# B&R Automation Studio project ABC_Pltzr
Automation Studio 

## Configuration PPC70_JOB24025

### Config.mpfilemanagerui - 4PPC70_101G_20F005/mapp/Config.mpfilemanagerui
```
Element gMpLinkMpFileManagerUI (Type=mpfilemanagerui)
```

## Logical view

Binary libraries used (declarations not repeated): AsBrStr, AsTCP, FileIO

### 1stReadme-ConfigAndRecipes.txt
```
Package name:
=============
appConfigAndRecipes

Desription:
===========
Package contains support for application wide Configuration and Recipe handling.

About:
======

Dependencies:
=============
- B&R Libraries: FileIO
- Other: bglib C utilities

Usage:
======
IMPORTANT: Make sure that the package is always located as a LAST item in the logical view!!!
This limitation is due to the compilatoin dependency and references to user defined structures defined
elsewhere and utilized here.

Examples:
=============
TODO
```

### MachineIO.typ
```iecst
(********************************************************************

 * COPYRIGHT -- Piedmont Automation Inc.

 ********************************************************************

 * File: MachineIO.typ

 * Author: goran

 * Created: Jun 1, 2015

 ********************************************************************

 *)
(*********************************************************************************

Machine IO Structure

*********************************************************************************)

TYPE
	machineIO_typ : 	STRUCT
		din : machineDI_typ;
		dout : machineDO_typ;
	END_STRUCT;
END_TYPE

(*********************************************************************************

	Machine Digital Inputs

*********************************************************************************)

TYPE
	machineDI_typ : 	STRUCT
		MCR : BOOL; (*Master Control Relay Energized*)
		Guard_DS1 : BOOL; (*Guard 1 Open DS1 # GUARD DOOR INSERTER*)
		Guard_DS2 : BOOL; (*Guard 2 Open DS2 # GUARD DOOR GROUPING RIGHT*)
		Guard_DS3 : BOOL; (*Guard 3 Open DS3 # GUARD DOOR DISPENSER*)
		Guard_DS4 : BOOL; (*Guard 4 Open DS4 # GUARD DOOR GROUPING LEFT*)
		Guard_DS5 : BOOL; (*Guard 5 Open DS5 # TBD*)
		Guard_DS6 : BOOL; (*Guard 6 Open DS6 # TBD*)
		EStop_PB1 : BOOL; (*EStop status 1 - PB1 - Enclosure*)
		EStop_PB2 : BOOL; (*EStop status 2 - PB2 - Infeed*)
		EStop_PB3 : BOOL; (*EStop status 3 - PB3 - Dispenser*)
		EStop_PB4 : BOOL; (*EStop status 4 - PB 4 - HMI*)
		EStop_PB5 : BOOL; (*EStop status 5 - PB5 - TBD*)
		EStop_PB6 : BOOL; (*EStop status 6 - PB6 - TBD*)
		MotorOverloads_OL : BOOL; (*MotorOverloads*)
		CustomerDischargeEnable_CR6 : BOOL; (*Customer Discharge Enable*)
		AirPressureSwitch_APS : BOOL; (*Air Pressure Switch APS*)
		PalletMagazineControl_SS2 : BOOL; (*Pallet Dispenser in Run Mode SS2*)
		PalleteDischLightCurtain_OSSD1 : BOOL; (*Pallete Dispenser Light Curtain CH A*)
		PalleteDischLightCurtain_OSSD2 : BOOL; (*Pallete Dispenser Light Curtain CH B*)
		ElevatorDetectPalletLayerLF_EE1 : BOOL; (*Detect Layer On Pallet EE1*)
		ProductAtStage_EE4Phy : BOOL;
		ProductAtStage_EE4TmrOn : TON;
		ProductAtStage_EE4TmrOf : TOF;
		ProductAtStage_EE4 : BOOL; (*Product/Case at Stage Position*)
		ElevatorDetectPalletLayerRT_EE3 : BOOL; (*Detect Layer On Pallet 2nd Eye EE3*)
		ZZZZZZZZZZZZZZZZZZZZZZZZZZZ : USINT;
		ElevatorFullUp_PR1 : BOOL; (*Elevator Full Up PR1*)
		ElevatorFullDown_PR2 : BOOL; (*Elevator Full Down PR2*)
		ElevatorAtGroupingRaise_PR4 : BOOL; (*Elevator @ Level for Raise PR4*)
		ElevatorAtGroupingLower_PR3 : BOOL; (*Elevator @ Level for Lower PR3*)
		ElevatorStopBlockRT_PR34 : BOOL; (*Elevator Stop Block Right Is Clear PR34*)
		ElevatorStopBlockLF_PR33 : BOOL; (*Elevator Stop Block Left Is Clear PR33*)
		ElevatorChainSlackRT_LS8 : BOOL; (*Elevator Chain Slack Right LS8*)
		ElevatorChainSlackLF_LS7 : BOOL; (*Elevator Chain Slack Left LS7*)
		TransferTableAtGrouping_PR6 : BOOL; (*Transfer Table At Grouping Side PR6*)
		TransferTableAtPallete_PR5 : BOOL; (*Table at Pallet Side PR5*)
		LayerStopBarDown_PR8 : BOOL; (*Layer Stop Bar/Stripper Bar is Down PR8*)
		LayerStopBarUp_PR7 : BOOL; (*Layer Stop Bar/Stripper Bar is Up PR7*)
		ProductAtInfeed_EE2Phy : BOOL; (*Product At Infeed Case / Counter EE2*)
		ProductAtInfeed_EE2TmrOn : TON; (*Product At Infeed Case / Counter EE2*)
		ProductAtInfeed_EE2TmrOf : TOF; (*Product At Infeed Case / Counter EE2*)
		ProductAtInfeed_EE2 : BOOL; (*Product At Infeed Case / Counter EE2*)
		RowTooLong_EE8Phy : BOOL;
		RowTooLong_EE8TmrOn : TON;
		RowTooLong_EE8TmrOf : TOF;
		RowTooLong_EE8 : BOOL; (*Comparison Count Row Too Long EE8*)
		RowPusherAtElevator_PR13 : BOOL; (*Row Pusher At Elevator PR13*)
		RowPusherReturned_PR11 : BOOL; (*Row Pusher Returned PR11*)
		PalletClawsAtTop_PR14 : BOOL; (*Pallet Dispenser at Top Position PR14*)
		PalletClawsAtMiddleLow_PR15 : BOOL; (*Pallet Dispenser Claws at Middle Position PR15*)
		PalletClawsAtMiddleHi_PR15A : BOOL; (*Pallet Claws at upper Middle*)
		PalletClawsAtBottom_PR16 : BOOL; (*Pallet Dispenser Claws at Bottom Position PR16*)
		PalletClawsClosedRT_PR18 : BOOL; (*Pallet Dispenser Right Claw Closed PR18*)
		PalletClawsClosedLF_PR20 : BOOL; (*Pallet Dispenser Left Claw Closed PR20*)
		PalletDispenserLowSupply_EE7 : BOOL; (*Pallet Dispenser Low Pallet Supply EE7*)
		PalletDispenserChainSlack_PR21 : BOOL; (*Pallet Dispenser Chain Slack PR21*)
		PalletDownOnDispenserCV_EE9 : BOOL; (*Pallet Dispenser Down on Dispenser Conveyor EE9*)
		ZZZZZZZZZZZZZZZZZZZZZZZZZZZ1 : USINT;
		Reset_PB : BOOL; (*Reset PushButton PB6*)
		PalletAtMachine_EE12 : BOOL; (*PalletAtMachine*)
		PalletAtDischarge_EE16 : BOOL; (*PalletAtDischarge*)
		Inserter_Control_In_Run_Mode : BOOL; (*Inserter Control in Run Mode SS3*)
		Inserter_Guard_Eye : BOOL; (*Inserter Guard Eye EE30*)
		Discharge_Guard_Eye : BOOL; (*Discharge Guard Eye EE5*)
		Pallet_On_Conveyor_2_After : BOOL; (*Pallet On Conveyor 2 After EE17*)
		Pallet_On_Conveyor_1_After : BOOL; (*Pallet On Conveyor 1 After EE16*)
		Drive1_Running : BOOL; (*Drive 1 Running VFD1*)
		Drive4_OverCurrent : BOOL; (*Drive 4 OverCurrent VFD4*)
		Motor_Protectors : BOOL; (*Motor Protectors OL*)
		Row_Pusher_At_PreGrouping : BOOL; (*Row Pusher At PreGrouping PR12*)
		Row_Pusher_Is_Down : BOOL; (*Row Pusher Is Down PR10*)
		Row_Pusher_Is_Up : BOOL; (*Row Pusher Is Up PR9*)
		MACHINE_ESTOPS_OK : BOOL; (*Machine ESTOPS*)
		ESTOPS_OK : BOOL; (*E-STOPS OKAY PB1*)
		Pallet_Chains_Are_Up : BOOL; (*Pallet Chains Are Up PR35*)
		Turn_Table_Is_Up_NOP : BOOL; (* TurnTable is Up-NOP PR23*)
		Turn_Table_Is_Down : BOOL; (* TurnTable is Down PR22*)
		Screen_Access : BOOL; (*Screen Access SS1*)
		AuxVFDsOk : BOOL; (*Auxiliar VFD's OK*)
		InserterAtMagazine : BOOL; (*Inserter At Magazine PR28*)
		InserterVacuumCupsIsDown : BOOL; (*Inserter Vacuum Cups Is Down PR27*)
		InserterIsDown : BOOL; (*Inserter is Down PR29*)
		InserterTierSheetBeltSlack : BOOL; (*Inserter Tier Sheet Belt Slack *)
		InserterLowTierSheetLevel : BOOL; (*Low Tier Sheet Level EE10*)
		InserterIsUp : BOOL; (*Inserter is Up PR26*)
		InserterSheetHeld : BOOL; (*Inserter Tier Sheet Held EE15*)
		Turn_Table_CW_Stop_Position : BOOL; (*Turn Table CW Stop Position PR24*)
	END_STRUCT;
END_TYPE

(*********************************************************************************

	Machine Digital Outputs

*********************************************************************************)

TYPE
	machineDO_typ : 	STRUCT
		MachineFaultBeacon_LT1 : BOOL; (*Machine Fault Beacon LT1*)
		MachineOkBeacon_LT2 : BOOL; (*Machine OK Beacon LT2*)
		PalletLowSupplyBeacon_LT3 : BOOL; (*Pallet Low Supply Beacon Light LT3*)
		LayerStopBarRaise_M3F : BOOL; (*Layer Bar Raise M3F*)
		LayerStopBarLower_M3R : BOOL; (*Layer Bar Lower M3R*)
		RowFormingRollers_M5 : BOOL; (*Grouping Rollers M5*)
		ProductInfeedCV_M6 : BOOL; (*Product Infeed Belt M6*)
		PalletDispenserCV_M7 : BOOL; (*Pallet Dispenser Conveyor M7*)
		PalletDispenserRaise_M8F : BOOL; (*Pallet Dispenser Raise M8F*)
		PalletDispenserLower_M8R : BOOL; (*Pallet Dispenser Lower M8R*)
		CustomerMachineRunning_CR4 : BOOL; (*Customer Facing Machine Running CR4*)
		CustomerMachineRunning_CR5 : BOOL; (*Customer Facing Machine Running CR5*)
		AirDump_SOL0 : BOOL; (*Air Dump SOL0*)
		TransferTableToGrouping_M2R : BOOL; (*Transfer Table To Grouping M2R*)
		TransferTableToPallet_M2F : BOOL; (*Transfer Table To Pallet M2F*)
		RowPusherReturn_M4R : BOOL; (*VFD4 REV*)
		RowPusherForward_M4F : BOOL; (*VFD4 FWD*)
		PalletClawsOpen_SOL7B : BOOL; (*Open Pallet Dispenser Claws SOL7B*)
		PalletClawsClose_SOL7A : BOOL; (*Close Pallet Dispenser Claws SOL7A*)
		FrontSquaringRetract_SOL11B : BOOL; (*End/Front Squaring Retract SOL11B*)
		FrontSquaringExtend_SOL11A : BOOL; (*End/Front Squaring Extend SOL11A*)
		SideSquaringRetract_SOL8B : BOOL; (*Side Squaring Retract SOL8B*)
		SideSquaringExtend_SOL8A : BOOL; (*Side Squaring Extend SOL8A*)
		BladeStop1Up_SOL3A : BOOL; (*Blade Stop 1 Lower SOL3B*)
		BladeStop1Dw_SOL3B : BOOL; (*Blade Stop 1 Raise SOL3A*)
		BladeStop2Up_SOL4A : BOOL; (*Blade Stop 1 Lower SOL3B*)
		BladeStop2Dw_SOL4B : BOOL; (*Blade Stop 1 Raise SOL3A*)
		BladeStop3Up_SOL5A : BOOL; (*Blade Stop 1 Lower SOL3B*)
		BladeStop3Dw_SOL5B : BOOL; (*Blade Stop 1 Raise SOL3A*)
		BladeStop4Up_SOL6A : BOOL; (*Blade Stop 1 Lower SOL3B*)
		BladeStop4Dw_SOL6B : BOOL; (*Blade Stop 1 Raise SOL3A*)
		BladeStop5Up_SOL13A : BOOL; (*Blade Stop 1 Lower SOL3B*)
		BladeStop5Dw_SOL13B : BOOL; (*Blade Stop 1 Raise SOL3A*)
		BladeStop6Up_SOL14A : BOOL; (*Blade Stop 1 Lower SOL3B*)
		BladeStop6Dw_SOL14B : BOOL; (*Blade Stop 1 Raise SOL3A*)
		CaseTurnerLower_SOL2B : BOOL; (*Case Turner Lower SOL2B*)
		CaseTurnerRaise_SOL2A : BOOL; (*Case Turner Raise SOL2A*)
		ZZZZZZZZZZZZZZZZZZZZZZZZZZZ : USINT;
		Full_Pallet_Conveyor : BOOL; (*Full Pallet Conveyor #VFD11FWD*)
		Full_Pallet_Conveyor_1_After : BOOL; (*Full Pallet Conveyor 1 After VFD12 # VFD12 FWD*)
		InserterHorizontalBrakeRelay : BOOL; (*Inserter Horizontal Brake Relay*)
		InserterVerticalBrakeRelay : BOOL; (*Inserter Vertical Brake Relay*)
		ElevatorSlow : BOOL; (*VFD1 DI2*)
		ElevatorRaise : BOOL; (*VFD1 FWD*)
		ElevatorLower : BOOL; (*VFD1 REV*)
		ElevatorFast : BOOL; (*VFD1 D1*)
		RowPusherFast : BOOL; (*VFD4 DI1*)
		VFD1BrakeRelay : BOOL; (*VFD1 Brake Relay CR1*)
		BladeStop4Lower : BOOL; (*Blade Stop 4 Lower SV6B*)
		BladeStop4Raise : BOOL; (*Blade Stop 4 Raise SV6A*)
		BladeStop3Lower : BOOL; (*Blade Stop 3 Lower SV5B*)
		BladeStop3Raise : BOOL; (*Blade Stop 3 Raise SV5A*)
		BladeStop2Lower : BOOL; (*Blade Stop 2 Lower SV4B*)
		BladeStop2Raise : BOOL; (*Blade Stop 2 Raise SV4A*)
		RowPusherLower : BOOL; (*Row Pusher Lower SV1B*)
		RowPusherRaise : BOOL; (*Row Pusher Raise SV1A*)
		VFD4BrakeRelay : BOOL; (*VFD4 Brake Relay CR2*)
		SheetInserterToPalletizer : BOOL; (*Sheet Inserter To Palletizer VFD10 REV*)
		SheetInserterHorizontalFastSpeed : BOOL; (*Sheet Inserter Horizontal Fast Speed VFD10 DI1*)
		SheetInserterRaise : BOOL; (*Sheet Inserter Raise VFD9 REV*)
		SheetInserterLower : BOOL; (*Sheet Inserter Lower VFD9 FWD*)
		SheetInserterVerticalSlowSpeed : BOOL; (*Sheet Inserter Vertical Slow Speed VFD9 DI1*)
		SheetInserterLockout : BOOL; (*Sheet Inserter Lockout SV9*)
		SheetInserterVacuum : BOOL; (*Sheet Inserter Vacuum SV10*)
		SheetInserterToMagazine : BOOL; (*Sheet Inserter To Magazine VFD10 FWD*)
		PalletChainsLower : BOOL; (*Pallet Chains Lower SV12B*)
		PalletChainsRaise : BOOL; (*Pallet Chains Raise SV12A*)
		CustomerPalletDischargingSignal : BOOL; (*Customer Pallet Discharging Signal CR5*)
		BladeStop6Lower : BOOL; (*Blade Stop 6 Lower SOL14B*)
		BladeStop6Raise : BOOL; (*Blade Stop 6 Raise SOL14A*)
		BladeStop5Lower : BOOL; (*Blade Stop 5 Lower SV13B*)
		BladeStop5Raise : BOOL; (*Blade Stop 5 Raise SV13A*)
		GroupingRollersSlowSpeed : BOOL; (*GroupingRollersSlowSpeed*)
	END_STRUCT;
END_TYPE

(**)
```

### Alarms.var
```iecst
(*********************************************************************************
 * Copyright: Piedmont Automation Inc
 * Author:    Goran
 * Created:   Jun 26, 2015/11:38 AM
 *********************************************************************************
 * Declaration of global variables
 *********************************************************************************)
VAR
	gAlarms : applicationAlarms_typ := (0);
	gAlarmsFiltered : applicationAlarms_typ := (0);
END_VAR
```

### ConfigApp.var
```iecst
(********************************************************************
 * COPYRIGHT --
 ********************************************************************
 * Package: ConfigAndRecipes
 * File: ConfigAndRecipes.var
 * Author: goran_2
 * Created: August 06, 2011
 ********************************************************************
 * Variables of package ConfigAndRecipes
 ********************************************************************)
VAR RETAIN
	gConfigApp : configApp_typ := (0); (*Application (Machine) Specific Configuration Data*)
END_VAR
```

- listItems.clm (not shown)

- paiCMRightMenu.clm (not shown)

- shiftStatus.clm (not shown)

- stationStatus.clm (not shown)

- Arial9pxValue.fninfo (not shown)

- DateTime.fninfo (not shown)

- MpHeader.fninfo (not shown)

- MpHtml_SDM.fninfo (not shown)

- alertMsg.layer (not shown)

- dialogMsg.layer (not shown)

- MpBackground.layer (not shown)

- paiHMIPvListView.layer (not shown)

- paiMpRecipeCustom1.layer (not shown)

- AlphaPadQVGA.tpr (not shown)

- vssver.scc (binary file, 48 bytes)
- vssver.scc (binary file, 48 bytes)
### EthSock.var
```iecst
(********************************************************************
 * COPYRIGHT (C) BERNECKER + RAINER, AUSTRIA, A-5142 EGGELSBERG
 ********************************************************************
 * Library: EthSock
 * File: EthSock.var
 * Created: 11.11.2003
 ********************************************************************
 * Constants of library EthSock
 ********************************************************************)
VAR CONSTANT
	ERR_ETH_ADDRNOTAVAIL	: UINT	:= 27149;
	ERR_ETH_TOOMANYREFS	: UINT	:= 27159;
	ERR_ETH_PROTONOTSUP	: UINT	:= 27143;
	ERR_ETH_NAMETOOLONG	: UINT	:= 27126;
	ERR_ETH_HOSTUNREACH	: UINT	:= 27165;
	ERR_ETH_DESTADDRREQ	: UINT	:= 27140;
	ERR_ETH_CONNREFUSED	: UINT	:= 27161;
	ERR_ETH_CONNABORTED	: UINT	:= 27153;
	ETH_SOCK_SEQPACKET	: DINT	:= 5;
	ERR_ETH_WOULDBLOCK	: UINT	:= 27170;
	ERR_ETH_SOCKNOTSUP	: UINT	:= 27144;
	ERR_ETH_NOPROTOOPT	: UINT	:= 27142;
	ERR_ETH_NETUNREACH	: UINT	:= 27151;
	ERR_ETH_INPROGRESS	: UINT	:= 27168;
	ERR_ETH_FD_SETSIZE	: UINT	:= 27200;
	ETH_SO_ACCEPTCONN	: DINT	:= 2;
	ETH_INET_ADDR_LEN	: USINT	:= 18;
	ERR_ETH_PROTOTYPE	: UINT	:= 27141;
	ERR_ETH_CONNRESET	: UINT	:= 27154;
	ERR_ETH_ADDRINUSE	: UINT	:= 27148;
	ETH_SO_REUSEADDR	: DINT	:= 4;
	ETH_SO_OOBINLINE	: DINT	:= 256;
	ETH_SO_KEEPALIVE	: DINT	:= 8;
	ETH_SO_DONTROUTE	: DINT	:= 16;
	ETH_SO_BROADCAST	: DINT	:= 32;
	ETH_IPPROTO_IGMP	: DINT	:= 2;
	ETH_IPPROTO_ICMP	: DINT	:= 1;
	ETH_AF_APPLETALK	: DINT	:= 16;
	ERR_ETH_TIMEDOUT	: UINT	:= 27160;
	ERR_ETH_SHUTDOWN	: UINT	:= 27158;
	ERR_ETH_PFNOTSUP	: UINT	:= 27146;
	ERR_ETH_OPNOTSUP	: UINT	:= 27145;
	ERR_ETH_NOTEMPTY	: UINT	:= 27115;
	ERR_ETH_NETRESET	: UINT	:= 27152;
	ERR_ETH_HOSTDOWN	: UINT	:= 27167;
	ERR_ETH_CANCELED	: UINT	:= 27172;
	ERR_ETH_AFNOTSUP	: UINT	:= 27147;
	ETH_SO_SNDTIMEO	: DINT	:= 4101;
	ETH_SO_SNDLOWAT	: DINT	:= 4099;
	ETH_SO_RCVTIMEO	: DINT	:= 4102;
	ETH_SO_RCVLOWAT	: DINT	:= 4100;
	ETH_SOCK_STREAM	: DINT	:= 1;
	ETH_IPPROTO_UDP	: DINT	:= 17;
	ETH_IPPROTO_TCP	: DINT	:= 6;
	ETH_IPPROTO_RAW	: DINT	:= 255;
	ETH_IPPROTO_PUP	: DINT	:= 12;
	ETH_IPPROTO_MAX	: DINT	:= 256;
	ETH_IPPROTO_IDP	: DINT	:= 17;
	ETH_IPPROTO_GGP	: DINT	:= 3;
	ERR_ETH_UNKNOWN	: UINT	:= 27249;
	ERR_ETH_NOTSOCK	: UINT	:= 27150;
	ERR_ETH_NOTCONN	: UINT	:= 27157;
	ERR_ETH_NETDOWN	: UINT	:= 27162;
	ERR_ETH_MSGSIZE	: UINT	:= 27136;
	ERR_ETH_ALREADY	: UINT	:= 27169;
	ETH_SOL_SOCKET	: DINT	:= 65535;
	ETH_SOCK_DGRAM	: DINT	:= 2;
	ETH_IPPROTO_IP	: DINT	:= 0;
	ETH_INADDR_ANY	: DINT	:= 0;
	ETH_FD_SETSIZE	: DINT	:= 256;
	ETH_AF_IMPLINK	: DINT	:= 3;
	ETH_AF_DATAKIT	: DINT	:= 9;
	ERR_ETH_TXTBSY	: UINT	:= 27163;
	ERR_ETH_NOTSUP	: UINT	:= 27135;
	ERR_ETH_NOTDIR	: UINT	:= 27120;
	ERR_ETH_NOTBLK	: UINT	:= 27166;
	ERR_ETH_NOEXEC	: UINT	:= 27108;
	ERR_ETH_NODATA	: UINT	:= 27178;
	ERR_ETH_NOBUFS	: UINT	:= 27155;
	ERR_ETH_ISCONN	: UINT	:= 27156;
	ERR_ETH_DEADLK	: UINT	:= 27133;
	ERR_ETH_BADMSG	: UINT	:= 27177;
	ERR_ETH_ACCESS	: UINT	:= 27113;
	ETH_SO_SNDBUF	: DINT	:= 4097;
	ETH_SO_RCVBUF	: DINT	:= 4098;
	ETH_SO_LINGER	: DINT	:= 128;
	ETH_SOMAXCONN	: DINT	:= 5;
	ETH_AF_UNSPEC	: DINT	:= 0;
	ETH_AF_HYLINK	: DINT	:= 15;
	ETH_AF_DECNET	: DINT	:= 12;
	ERR_ETH_SPIPE	: UINT	:= 27129;
	ERR_ETH_RANGE	: UINT	:= 27138;
	ERR_ETH_PROTO	: UINT	:= 27176;
	ERR_ETH_NOTTY	: UINT	:= 27125;
	ERR_ETH_NOSYS	: UINT	:= 27171;
	ERR_ETH_NOSTR	: UINT	:= 27175;
	ERR_ETH_NOSPC	: UINT	:= 27128;
	ERR_ETH_NOMSG	: UINT	:= 27180;
	ERR_ETH_NOMGR	: UINT	:= 27248;
	ERR_ETH_NOMEM	: UINT	:= 27112;
	ERR_ETH_NOLCK	: UINT	:= 27134;
	ERR_ETH_NOENT	: UINT	:= 27102;
	ERR_ETH_NODEV	: UINT	:= 27119;
	ERR_ETH_NFILE	: UINT	:= 27123;
	ERR_ETH_MLINK	: UINT	:= 27131;
	ERR_ETH_MFILE	: UINT	:= 27124;
	ERR_ETH_ISDIR	: UINT	:= 27121;
	ERR_ETH_INVAL	: UINT	:= 27122;
	ERR_ETH_FAULT	: UINT	:= 27114;
	ERR_ETH_EXIST	: UINT	:= 27117;
	ERR_ETH_CHILD	: UINT	:= 27110;
	ERR_ETH_AGAIN	: UINT	:= 27111;
	ETH_SO_ERROR	: DINT	:= 4103;
	ETH_SO_DEBUG	: DINT	:= 1;
	ETH_SOCK_RDM	: DINT	:= 4;
	ETH_SOCK_RAW	: DINT	:= 3;
	ETH_FIONREAD	: DINT	:= 1;
	ETH_AF_CHAOS	: DINT	:= 5;
	ETH_AF_CCITT	: DINT	:= 10;
	ERR_ETH_XDEV	: UINT	:= 27118;
	ERR_ETH_TIME	: UINT	:= 27179;
	ERR_ETH_SRCH	: UINT	:= 27103;
	ERR_ETH_ROFS	: UINT	:= 27130;
	ERR_ETH_PIPE	: UINT	:= 27132;
	ERR_ETH_PERM	: UINT	:= 27101;
	ERR_ETH_NXIO	: UINT	:= 27106;
	ERR_ETH_NOSR	: UINT	:= 27174;
	ERR_ETH_LOOP	: UINT	:= 27164;
	ERR_ETH_INTR	: UINT	:= 27104;
	ERR_ETH_FBIG	: UINT	:= 27127;
	ERR_ETH_BUSY	: UINT	:= 27116;
	ERR_ETH_BASE	: UINT	:= 27100;
	ERR_ETH_BADF	: UINT	:= 27109;
	ERR_ETH_2BIG	: UINT	:= 27107;
	ETH_SO_TYPE	: DINT	:= 4104;
	ETH_FIONBIO	: DINT	:= 16;
	ETH_AF_UNIX	: DINT	:= 1;
	ETH_AF_INET	: DINT	:= 2;
	ETH_AF_ECMA	: DINT	:= 8;
	ERR_ETH_MAX	: UINT	:= 27181;
	ERR_ETH_DOM	: UINT	:= 27137;
	ETH_AF_SNA	: DINT	:= 11;
	ETH_AF_PUP	: DINT	:= 4;
	ETH_AF_OSI	: DINT	:= 7;
	ETH_AF_LAT	: DINT	:= 14;
	ETH_AF_ISO	: DINT	:= 7;
	ETH_AF_DLI	: DINT	:= 13;
	ERR_SOCKET	: DINT	:= -1;
	ERR_ETH_IO	: UINT	:= 27105;
	ETH_AF_NS	: DINT	:= 6;
END_VAR
```

### MpAlarmError.typ
```iecst
TYPE
    MpAlarmErrorEnum :
        ( (* Error numbers of library MpAlarm *)
        mpALARM_NO_ERROR := 0, (* No error *)
        mpALARM_ERR_ACTIVATION := -1064239103, (* Could not create component [Error: 1, 0xc0910001] *)
        mpALARM_ERR_MPLINK_NULL := -1064239102, (* MpLink is NULL pointer [Error: 2, 0xc0910002] *)
        mpALARM_ERR_MPLINK_INVALID := -1064239101, (* MpLink connection not allowed [Error: 3, 0xc0910003] *)
        mpALARM_ERR_MPLINK_CHANGED := -1064239100, (* MpLink modified [Error: 4, 0xc0910004] *)
        mpALARM_ERR_MPLINK_CORRUPT := -1064239099, (* Invalid MpLink contents [Error: 5, 0xc0910005] *)
        mpALARM_ERR_MPLINK_IN_USE := -1064239098, (* MpLink already in use [Error: 6, 0xc0910006] *)
        mpALARM_ERR_CONFIG_INVALID := -1064239091, (* Invalid Configuration [Error: 13, 0xc091000d] *)
        mpALARM_ERR_ALARM_ID_OVER_MAX := -1064157184, (* Alarm number too high [Error: 16384, 0xc0924000] *)
        mpALARM_ERR_IMAGE_NULL := -1064157183, (* Image is NULL [Error: 16385, 0xc0924001] *)
        mpALARM_WRN_IMAGE_SIZE := -2137899006, (* Image smaller than maximum numbers of alarms [Warning: 16386, 0x80924002] *)
        mpALARM_ERR_NO_ALARMS_FOUND := -1064157181, (* Component has no alarms [Error: 16387, 0xc0924003] *)
        mpALARM_ERR_NUMBER_OF_ALARMS := -1064157180, (* Invalid number of alarms [Error: 16388, 0xc0924004] *)
        mpALARM_INF_WAIT_BASIC_FB := 1083326469 (* Waiting for parent component [Informational: 16389, 0x40924005] *)
        );
END_TYPE
```

### MpCom.typ
```iecst
TYPE
	MpComFacilitiesEnum :
		(
		mpCOM_FAC_UNDEFINED := -1, (*No active error*)
		mpCOM_FAC_ARCORE := 0, (*Facility for legacy error code from AR libraries in UINT format*)
		mpCOM_FAC_SAFETY1 := 1, (*Safety facility*)
		mpCOM_FAC_SAFETY2 := 2, (*Safety facility*)
		mpCOM_FAC_GMC1 := 96, (*GMC facility*)
		mpCOM_FAC_GMC2 := 97, (*GMC facility*)
		mpCOM_FAC_GMCAXIS := 98, (*GMC Axis facility*)
		mpCOM_FAC_GMCAXESGROUP := 99, (*GMC Axes group facility*)
		mpCOM_FAC_GMCARNCGROUP := 103, (*GMC Arnc group facility*)
		mpCOM_FAC_TRF := 105, (*TRF facility*)
		mpCOM_FAC_MAPP_INTERNAL := 144, (*mapp Internal Facility*)
		mpCOM_FAC_MAPP_CORE := 145, (*mapp Core Facility*)
		mpCOM_FAC_MAPP_INFRASTRUCTURE := 146, (*mapp Infrastructure Facility*)
		mpCOM_FAC_MAPP_MECHATRONIC := 147, (*mapp Mechatronics Facility*)
		mpCOM_FAC_MAPP_INDUSTRY := 148 (*mapp Industry Facility*)
		);
	MpComConfigScopeEnum :
		(
		mpCOM_CONFIG_SCOPE_COMPONENT := 0, (*Import / Export configuration only for given component*)
		mpCOM_CONFIG_SCOPE_BRANCH := 1 (*Import / Export configuration for given component and all its sub-components*)
		);
	MpComInternalIDType : 	STRUCT
		ID : DINT; (*Status ID*)
		Severity : MpComSeveritiesEnum; (*Status severity*)
		Facility : MpComFacilitiesEnum; (*Status facility*)
		Code : UINT; (*Status / Error code*)
	END_STRUCT;
	MpComStatusIDType : 	STRUCT
		ID : MpComErrorEnum; (*Status ID*)
		Severity : MpComSeveritiesEnum; (*Status severity*)
		Facility : MpComFacilitiesEnum; (*Status facility*)
		Code : UINT; (*Status / Error code*)
	END_STRUCT;
	MpComDiagType : 	STRUCT
		StatusID : MpComStatusIDType; (*StatusID diagnostic structure *)
	END_STRUCT;
	MpComConfigManagerInfoType : 	STRUCT
		Diag : MpComDiagType; (*Diagnostic structure for the status ID*)
	END_STRUCT;
	MpComIdentType : 	STRUCT
		Internal : ARRAY[0..1]OF UDINT; (*For internal use only*)
	END_STRUCT;
	MpComInternalDataType : 	STRUCT
		pObject : UDINT;
		State : UDINT;
	END_STRUCT;
	MpComConfigInternalType : 	STRUCT
		pObject : UDINT;
		State : DINT;
	END_STRUCT;
	MpComSeveritiesEnum :
		(
		mpCOM_SEV_SUCCESS := 0, (*Success - no error*)
		mpCOM_SEV_INFORMATIONAL := 1, (*Severity: Informational*)
		mpCOM_SEV_WARNING := 2, (*Severity: Warning*)
		mpCOM_SEV_ERROR := 3 (*Severity: Error*)
		);
	MpComDumpInternalType : 	STRUCT
		CmdOld : BOOL;
	END_STRUCT;
	MpComLoggerUISetupType : 	STRUCT
		LoggerListSize : UINT := 20; (*Number of logger entries to be displayed on one page of the list in the HMI application*)
		LoggerScrollWindow : USINT := 0; (*Determines how many entries from the list are displayed in advance when scrolling up and down*)
	END_STRUCT;
	MpComLoggerUIConnectType : 	STRUCT
		Status : MpComLoggerUIStatusEnum;
		List : MpComLoggerUILoggerListType; (*List of resultant logger entries*)
		Clear : BOOL; (*Clean the internal buffer*)
		SearchFilter : STRING[255]; (*Filter used to define the visibility of entries*)
	END_STRUCT;
	MpComLoggerUIStatusEnum :
		(
		mpCOM_LOGGERUI_IDLE := 0,
		mpCOM_LOGGERUI_REFRESH := 1,
		mpCOM_LOGGERUI_ERROR := 2
		);
	MpComLoggerUILoggerListType : 	STRUCT
		Message : ARRAY[0..19]OF STRING[255]; (*List of logger entries: message*)
		StatusID : ARRAY[0..19]OF DINT; (*List of logger entries: status ID*)
		ErrorNumber : ARRAY[0..19]OF UINT; (*List of logger entries: error code as part of Status ID*)
		Time : ARRAY[0..19]OF MpComLoggerUIDateTimeType; (*List of logger entries: date, time and microseconds*)
		Component : ARRAY[0..19]OF STRING[50]; (*List of logger entries: component name*)
		Facility : ARRAY[0..19]OF MpComFacilitiesEnum; (*List of logger entries: facility as part of Status ID*)
		Severity : ARRAY[0..19]OF MpComSeveritiesEnum; (*List of logger entries: severity as part of Status ID*)
		PageUp : BOOL; (*Jumps to the start of the current page and then scrolls up one page at a time *)
		PageDown : BOOL; (*Jumps to the end of the current page and then scrolls down one page at a time *)
		StepUp : BOOL; (*Selects the previous entry in the list*)
		StepDown : BOOL; (*Selects the next entry in the list*)
		RangeStart : REAL; (*Shows a bar indicating which part of the list is currently being displayed-Start [%]*)
		RangeEnd : REAL; (*Shows a bar indicating which part of the list is currently being displayed-End [%]*)
	END_STRUCT;
	MpComLoggerUIDateTimeType : 	STRUCT
		DateTime : DATE_AND_TIME; (*List of logger entries: date and time: the view could be customized on VC*)
		Microseconds : UDINT; (*List of logger entries: additional information about microseconds when the event was triggered*)
	END_STRUCT;
	MpComLoggerUIInfoType : 	STRUCT
		CurrentBufferEntries : UINT; (*Number of entries currently in the internal buffer. It is a ring buffer, it means that reached the BufferSize it doesn't increase any more*)
		Diag : MpComDiagType; (*Diagnostic structure for the status ID*)
	END_STRUCT;
END_TYPE
```

- vssver.scc (binary file, 48 bytes)
### appDraw.var
```iecst
VAR RETAIN
	gTestLayer : ARRAY[0..9] OF appControlAnimationRow_typ;
END_VAR
VAR
	gDrawRect : ARRAY[0..PADRAW_RECT_MAXIDX] OF paDrawRect_typ;
	gDrawBoxLayer : paDrawBoxDrawing_typ;
	gCamApp : paCamEditApp_typ;
END_VAR
VAR RETAIN
	gBoxSize : paDrawBoxSize_typ;
END_VAR
```

### Program Logical/MachineControl/caseturner

#### Cyclic.ld
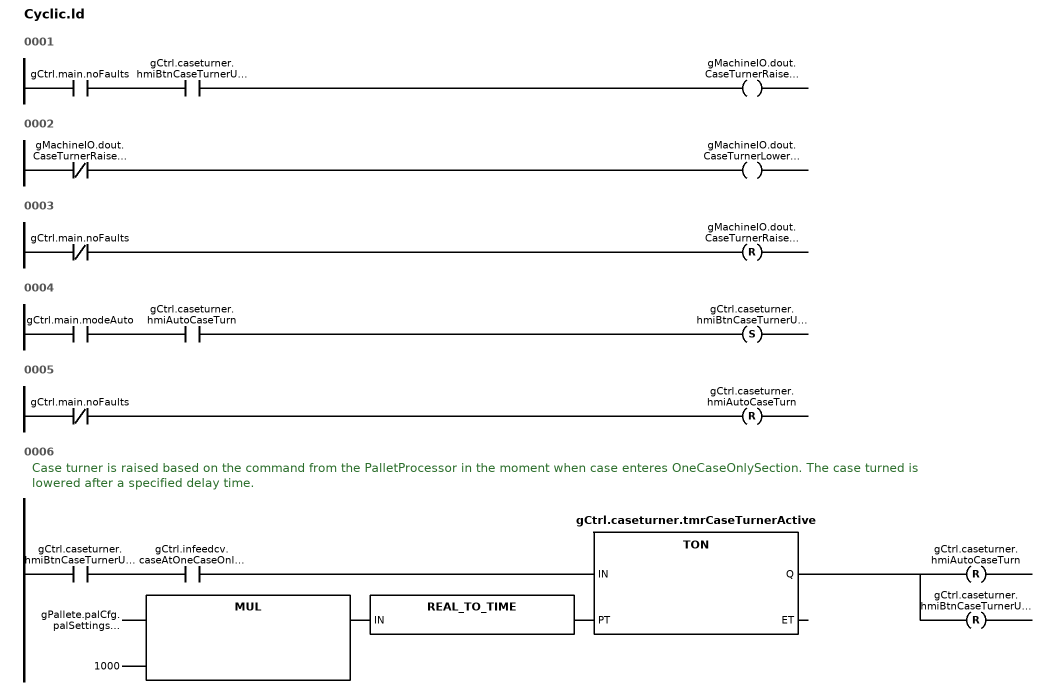
Ladder, written as Structured Text:
```iecst
PROGRAM _CYCLIC
VAR
    _p1 : BOOL;
END_VAR
(* Network 1 *)
gMachineIO.dout.CaseTurnerRaise_SOL2A := gCtrl.main.noFaults AND gCtrl.caseturner.hmiBtnCaseTurnerUpDown;

(* Network 2 *)
gMachineIO.dout.CaseTurnerLower_SOL2B := NOT gMachineIO.dout.CaseTurnerRaise_SOL2A;

(* Network 3 *)
IF NOT gCtrl.main.noFaults THEN gMachineIO.dout.CaseTurnerRaise_SOL2A := FALSE; END_IF;

(* Network 4 *)
IF gCtrl.main.modeAuto AND gCtrl.caseturner.hmiAutoCaseTurn THEN
    gCtrl.caseturner.hmiBtnCaseTurnerUpDown := TRUE;
END_IF;

(* Network 5 *)
IF NOT gCtrl.main.noFaults THEN gCtrl.caseturner.hmiAutoCaseTurn := FALSE; END_IF;

(* Network 6: Case turner is raised based on the command from the PalletProcessor in the moment when case enteres OneCaseOnlySection. The case turned is lowered after a specified delay time. *)
gCtrl.caseturner.tmrCaseTurnerActive(IN := gCtrl.caseturner.hmiBtnCaseTurnerUpDown AND gCtrl.infeedcv.caseAtOneCaseOnlySection, PT := REAL_TO_TIME(gPallete.palCfg.palSettings.timers.onTmCaseTurner * 1000));
_p1 := gCtrl.caseturner.tmrCaseTurnerActive.Q;
IF gCtrl.caseturner.tmrCaseTurnerActive.Q THEN gCtrl.caseturner.hmiAutoCaseTurn := FALSE; END_IF;
IF _p1 THEN gCtrl.caseturner.hmiBtnCaseTurnerUpDown := FALSE; END_IF;
END_PROGRAM
```

### Program Logical/MachineControl/elevmove

#### Cyclic.st
```iecst
PROGRAM _CYCLIC
	(* Insert code here *)

	//===========================================================================================
	//Manipulate elevator speeds (lower speed when approaching home position)
	IF gCtrl.main.elevatorStopBlockActive THEN
		//When stop blocks are active make sure that the elevator only moves using a slow speed!!!
		gMachineVFD[1].vfdCtrl.iVelocitySetPoint := DINT_TO_INT(gPallete.palCfg.palSettings.vfd[1].velocitySlow_rpm);
		IF gMachineVFD[1].vfdCtrl.iVelocitySetPoint > 300 THEN
			gMachineVFD[1].vfdCtrl.iVelocitySetPoint := 300;
		END_IF;
	ELSE
		IF gCtrl.elevator.hmiBtnElevatorToGrouping AND (gCtrl.elevator.elevatorIsAboveNearHome OR gCtrl.elevator.elevatorIsBelowNearHome) THEN
			gMachineVFD[1].vfdCtrl.iVelocitySetPoint := DINT_TO_INT(gPallete.palCfg.palSettings.vfd[1].velocitySlow_rpm);
		ELSE
			gMachineVFD[1].vfdCtrl.iVelocitySetPoint := DINT_TO_INT(gPallete.palCfg.palSettings.vfd[1].velocity_rpm);
		END_IF;

		//Any Jog move ALWAYS uses SLOW SPEED
		//In auto mode (i.e. hmiBtnElevatorRev) reverse mode ALWAYS uses SLOW SPEED when approaching pallet top (i.e. table is NOT at grouping)
		IF (NOT gCtrl.transfertable.isTableAtGrouping AND gCtrl.elevator.hmiBtnElevatorRev) OR
			( (gCtrl.elevator.elevatorIsBelowHome OR  gCtrl.elevator.elevatorIsBelowNearHome OR gCtrl.elevator.elevatorIsBelowHomeUnknown) AND (gCtrl.elevator.hmiBtnElevatorRevJog OR gCtrl.elevator.hmiBtnElevatorFwdJog) ) THEN
			gMachineVFD[1].vfdCtrl.iVelocitySetPoint := DINT_TO_INT(gPallete.palCfg.palSettings.vfd[1].velocitySlow_rpm);
		END_IF;

	END_IF;

	//===========================================================================================
	//Process request for: Move elevator to Grouping Position
	IF gCtrl.elevator.hmiBtnElevatorToGrouping THEN
		gCtrl.elevator.hmiBtnElevatorToPallete := 0;
		gCtrl.elevator.hmiBtnElevatorToAbovePallete := 0;
		gCtrl.elevator.hmiBtnElevatorToTop := 0;

		//reset hmiBtnElevatorToGrouping only when at home and vfd at stand still (avoid issue with long decel)
		IF gCtrl.elevator.elevatorIsAtHome AND (gMachineVFD[1].vfdIn.Status.CurrentVelocity = 0) THEN
			gCtrl.elevator.hmiBtnElevatorToGrouping := 0;
		END_IF;

		IF gCtrl.elevator.elevatorIsAtHome THEN
			//gCtrl.elevator.hmiBtnElevatorToGrouping := 0;
			gCtrl.elevator.hmiBtnElevatorRev := 0;
			gCtrl.elevator.hmiBtnElevatorFwd := 0;
		ELSE

			IF NOT gCtrl.transfertable.isTableAtGrouping THEN//tansfer table back to grouping before driving elveator up/down
				gCtrl.transfertable.hmiBtnTableRev := 1;
			END_IF;

			IF gCtrl.elevator.elevatorIsAboveHome THEN//above? > send it down
				gCtrl.elevator.hmiBtnElevatorFwd := 0;
				gCtrl.elevator.hmiBtnElevatorRev := 1;
			ELSIF gCtrl.elevator.elevatorIsBelowHome THEN//below> > send it up
				gCtrl.elevator.hmiBtnElevatorFwd := 1;
				gCtrl.elevator.hmiBtnElevatorRev := 0;
			ELSE //don't know > send it down ???? should not happen
				gCtrl.elevator.hmiBtnElevatorFwd := 0;
				gCtrl.elevator.hmiBtnElevatorRev := 1;
			END_IF;
		END_IF;
	END_IF

	//===========================================================================================
	//Process request for: Move elevator to top of the pallet position
	gCtrl.elevator.tmrPalletePEOn.PT := REAL_TO_TIME (gPallete.palCfg.palSettings.timers.onDlyEEPallete * 1000.0);
	gCtrl.elevator.tmrPalletePEOn.IN := gMachineIO.din.ElevatorDetectPalletLayerLF_EE1 OR gMachineIO.din.ElevatorFullDown_PR2;
	gCtrl.elevator.tmrPalletePEOn();

	gCtrl.elevator.tmrPalletePEOff.PT := REAL_TO_TIME (gPallete.palCfg.palSettings.timers.offDlyEEPallete * 1000.0);
	gCtrl.elevator.tmrPalletePEOff.IN := gMachineIO.din.ElevatorDetectPalletLayerLF_EE1;
	gCtrl.elevator.tmrPalletePEOff();

	//any move resets above pallete flags
	IF gCtrl.elevator.elevatorIsAtPalleteBelowHome AND (gCtrl.elevator.hmiBtnElevatorFwd OR gCtrl.elevator.hmiBtnElevatorRev) THEN
		//gCtrl.elevator.elevatorIsAtPalleteAboveHome := 0;//not used!!!
		gCtrl.elevator.elevatorIsAtPalleteBelowHome := 0;
	END_IF;

	//===========================================================================================
	IF (gCtrl.elevator.hmiBtnElevatorToPallete = 1) THEN
		gCtrl.elevator.hmiBtnElevatorToGrouping := 0;
		gCtrl.elevator.hmiBtnElevatorToAbovePallete := 0;
		gCtrl.elevator.hmiBtnElevatorToTop := 0;

		//Sequence starts here!
		IF (gCtrl.elevator.elevatorIsAtHome AND gCtrl.transfertable.isTableAtGrouping) THEN
			IF gMachineIO.din.ElevatorDetectPalletLayerLF_EE1 THEN
				//If pallete detect PE is blocked > move elevator up
				gCtrl.elevator.hmiBtnElevatorFwd := 1;
				gCtrl.elevator.hmiBtnElevatorRev := 0;
			ELSE
				//If pallete detect PE NOT blocked > move table to pallete
				gCtrl.transfertable.hmiBtnTableFwd := 1;
				gCtrl.transfertable.hmiBtnTableRev := 0;
			END_IF;
		END_IF;

		//monitor elevator up move
		IF gCtrl.elevator.hmiBtnElevatorFwd AND NOT gCtrl.elevator.tmrPalletePEOff.Q THEN
			//when elevator move up is complete > move the table to the pallete side
			gCtrl.elevator.hmiBtnElevatorFwd := 0;
			gCtrl.elevator.hmiBtnElevatorRev := 0;

			//If pallete detect PE NOT blocked > move table to pallete
			gCtrl.transfertable.hmiBtnTableFwd := 1;
			gCtrl.transfertable.hmiBtnTableRev := 0;
		END_IF;

		//when table at pallete > move elevator down
		IF gCtrl.transfertable.isTableAtPallete AND NOT gCtrl.elevator.hmiBtnElevatorRev THEN
			gCtrl.elevator.hmiBtnElevatorFwd := 0;
			gCtrl.elevator.hmiBtnElevatorRev := 1;
		END_IF;

		IF gCtrl.elevator.hmiBtnElevatorRev AND gCtrl.elevator.tmrPalletePEOn.Q THEN
			gCtrl.elevator.elevatorIsAtPalleteBelowHome := 1;//elevator is at pallet (same flag used for above home OR below home)
			gCtrl.elevator.hmiBtnElevatorFwd := 0;
			gCtrl.elevator.hmiBtnElevatorRev := 0;
			gCtrl.elevator.hmiBtnElevatorToPallete := 0;
		END_IF;

	END_IF;

	//===========================================================================================
	//Process request for: Move elevator to Above Pallete
	IF gCtrl.elevator.hmiBtnElevatorToAbovePallete THEN
		gCtrl.elevator.hmiBtnElevatorToPallete := 0;
		gCtrl.elevator.hmiBtnElevatorToGrouping := 0;
		gCtrl.elevator.hmiBtnElevatorToTop := 0;

		//Sequence starts here!
		IF gCtrl.transfertable.isTableAtGrouping THEN
			IF gMachineIO.din.ElevatorDetectPalletLayerLF_EE1 THEN
				//If pallete detect PE is blocked > move elevator up
				gCtrl.elevator.hmiBtnElevatorFwd := 1;
				gCtrl.elevator.hmiBtnElevatorRev := 0;
			END_IF;
		END_IF;

		//monitor elevator up move
		//IF gCtrl.elevator.hmiBtnElevatorFwd AND NOT gCtrl.elevator.tmrPalletePEOff.Q THEN
		IF NOT gCtrl.elevator.tmrPalletePEOff.Q THEN
			//when elevator move up is complete > move the table to the pallete side
			gCtrl.elevator.hmiBtnElevatorFwd := 0;
			gCtrl.elevator.hmiBtnElevatorRev := 0;
			gCtrl.elevator.hmiBtnElevatorToAbovePallete := 0;
		END_IF;

	END_IF;

	//===========================================================================================
	//Process request for: Move elevator to Top Most Position
	IF gCtrl.elevator.hmiBtnElevatorToTop THEN
		gCtrl.elevator.hmiBtnElevatorToPallete := 0;
		gCtrl.elevator.hmiBtnElevatorToGrouping := 0;
		gCtrl.elevator.hmiBtnElevatorToAbovePallete := 0;

		//Sequence starts here!
		IF gCtrl.transfertable.isTableAtGrouping THEN
			//If pallete detect PE is blocked > move elevator up
			gCtrl.elevator.hmiBtnElevatorFwd := 1;
			gCtrl.elevator.hmiBtnElevatorRev := 0;
		END_IF;

		//monitor elevator up move
		//IF gCtrl.elevator.hmiBtnElevatorFwd AND NOT gCtrl.elevator.tmrPalletePEOff.Q THEN
		IF gCtrl.elevator.elevatorIsAtTop THEN
			//when elevator move up is complete > move the table to the pallete side
			gCtrl.elevator.hmiBtnElevatorFwd := 0;
			gCtrl.elevator.hmiBtnElevatorRev := 0;
			gCtrl.elevator.hmiBtnElevatorToTop := 0;
		END_IF;

	END_IF;

	//===========================================================================================
	//In case of faults > reset move requests, stop the VFD-s
	IF NOT gCtrl.main.noFaults THEN
		gCtrl.elevator.hmiBtnElevatorToPallete := 0;
		gCtrl.elevator.hmiBtnElevatorToGrouping := 0;
		gCtrl.elevator.hmiBtnElevatorToAbovePallete := 0;
		gCtrl.elevator.hmiBtnElevatorFwd := 0;
		gCtrl.elevator.hmiBtnElevatorRev := 0;
	END_IF;

END_PROGRAM
```

### Program Logical/MachineControl/infcvidle

#### Cyclic.ld
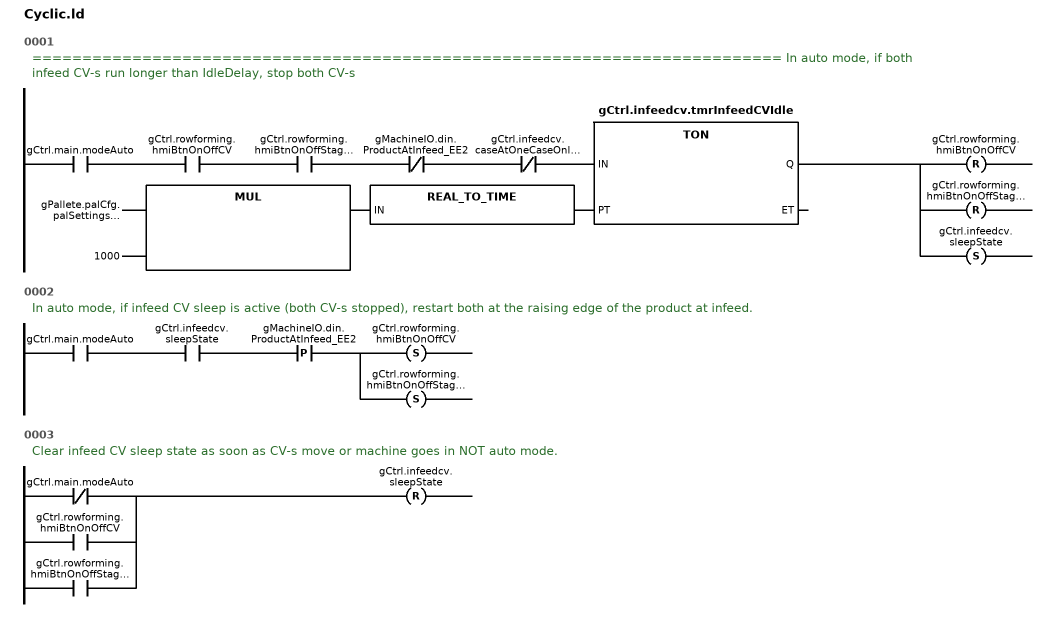
Ladder, written as Structured Text:
```iecst
PROGRAM _CYCLIC
VAR
    _p1 : BOOL;
    _e2 : R_TRIG;
    _p3 : BOOL;
END_VAR
(* Network 1: =========================================================================== In auto mode, if both infeed CV-s run longer than IdleDelay, stop both CV-s *)
gCtrl.infeedcv.tmrInfeedCVIdle(IN := gCtrl.main.modeAuto AND gCtrl.rowforming.hmiBtnOnOffCV AND gCtrl.rowforming.hmiBtnOnOffStageCV AND NOT gMachineIO.din.ProductAtInfeed_EE2 AND NOT gCtrl.infeedcv.caseAtOneCaseOnlySection, PT := REAL_TO_TIME(gPallete.palCfg.palSettings.timers.infeedCVIdleTime * 1000));
_p1 := gCtrl.infeedcv.tmrInfeedCVIdle.Q;
IF gCtrl.infeedcv.tmrInfeedCVIdle.Q THEN gCtrl.rowforming.hmiBtnOnOffCV := FALSE; END_IF;
IF _p1 THEN
    gCtrl.rowforming.hmiBtnOnOffStageCV := FALSE;
    gCtrl.infeedcv.sleepState := TRUE;
END_IF;

(* Network 2: In auto mode, if infeed CV sleep is active (both CV-s stopped), restart both at the raising edge of the product at infeed. *)
_e2(CLK := gMachineIO.din.ProductAtInfeed_EE2);
_p3 := gCtrl.main.modeAuto AND gCtrl.infeedcv.sleepState AND _e2.Q;
IF _p3 THEN
    gCtrl.rowforming.hmiBtnOnOffCV := TRUE;
    gCtrl.rowforming.hmiBtnOnOffStageCV := TRUE;
END_IF;

(* Network 3: Clear infeed CV sleep state as soon as CV-s move or machine goes in NOT auto mode. *)
IF NOT gCtrl.main.modeAuto OR gCtrl.rowforming.hmiBtnOnOffCV OR gCtrl.rowforming.hmiBtnOnOffStageCV THEN
    gCtrl.infeedcv.sleepState := FALSE;
END_IF;
END_PROGRAM
```

- Program Logical/MachineControl/palletinfdis (IEC) (no source held here)

### Program Logical/MachineControl/simonly

#### Cyclic.ld
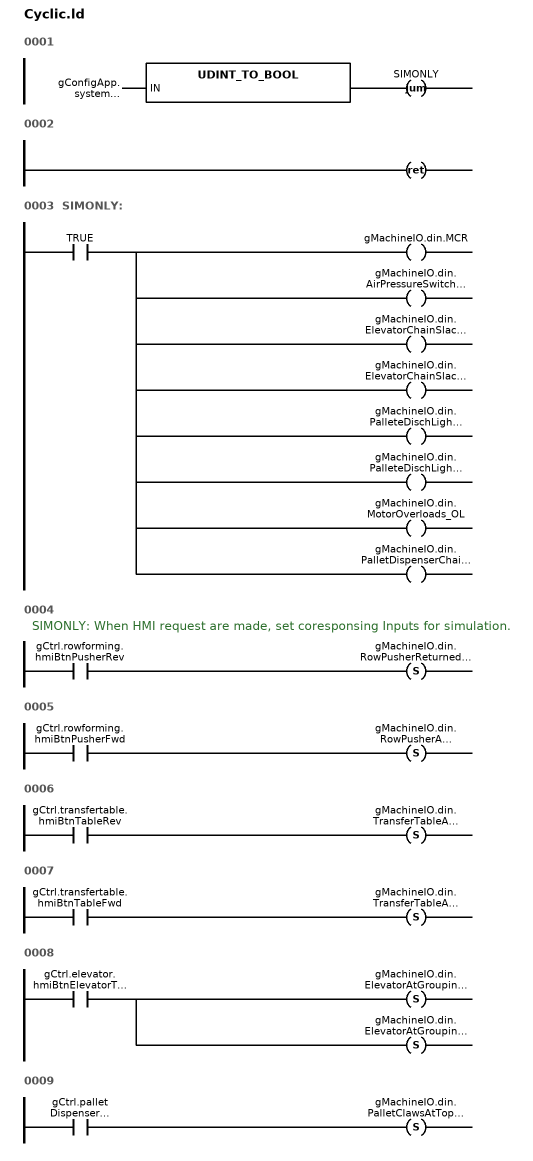
Ladder, written as Structured Text:
```iecst
PROGRAM _CYCLIC
(* Network 1 *)
IF UDINT_TO_BOOL(gConfigApp.system.simulationMode) THEN JMP SIMONLY; END_IF;

(* Network 2 *)
RETURN;

(* Network 3 *)
SIMONLY:
gMachineIO.din.MCR := TRUE;
gMachineIO.din.AirPressureSwitch_APS := TRUE;
gMachineIO.din.ElevatorChainSlackLF_LS7 := TRUE;
gMachineIO.din.ElevatorChainSlackRT_LS8 := TRUE;
gMachineIO.din.PalleteDischLightCurtain_OSSD1 := TRUE;
gMachineIO.din.PalleteDischLightCurtain_OSSD2 := TRUE;
gMachineIO.din.MotorOverloads_OL := TRUE;
gMachineIO.din.PalletDispenserChainSlack_PR21 := TRUE;

(* Network 4: SIMONLY: When HMI request are made, set coresponsing Inputs for simulation. *)
IF gCtrl.rowforming.hmiBtnPusherRev THEN gMachineIO.din.RowPusherReturned_PR11 := TRUE; END_IF;

(* Network 5 *)
IF gCtrl.rowforming.hmiBtnPusherFwd THEN gMachineIO.din.RowPusherAtElevator_PR13 := TRUE; END_IF;

(* Network 6 *)
IF gCtrl.transfertable.hmiBtnTableRev THEN gMachineIO.din.TransferTableAtGrouping_PR6 := TRUE; END_IF;

(* Network 7 *)
IF gCtrl.transfertable.hmiBtnTableFwd THEN gMachineIO.din.TransferTableAtPallete_PR5 := TRUE; END_IF;

(* Network 8 *)
IF gCtrl.elevator.hmiBtnElevatorToGrouping THEN
    gMachineIO.din.ElevatorAtGroupingLower_PR3 := TRUE;
    gMachineIO.din.ElevatorAtGroupingRaise_PR4 := TRUE;
END_IF;

(* Network 9 *)
IF gCtrl.palletDispenser.hmiBtnClawsLiftToTop THEN gMachineIO.din.PalletClawsAtTop_PR14 := TRUE; END_IF;
END_PROGRAM
```

### Program Logical/MachineControl/squaring

#### Cyclic.ld
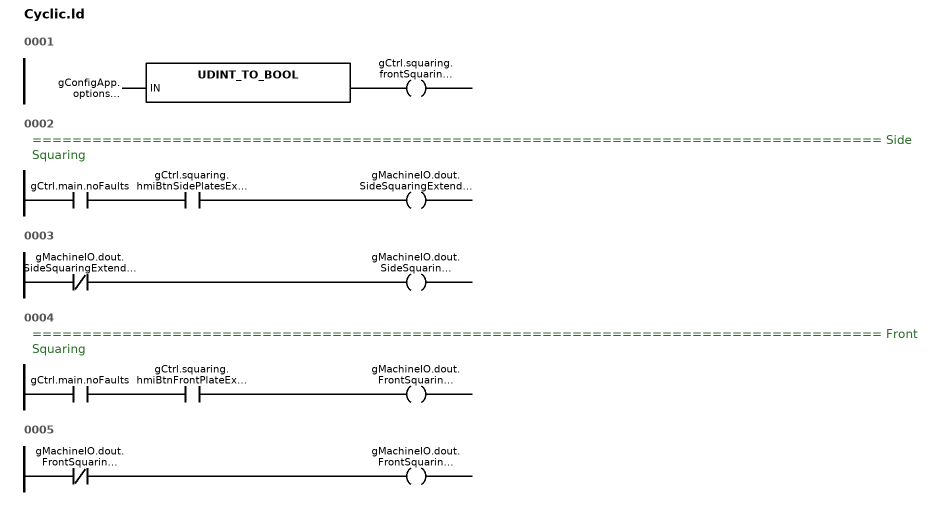
Ladder, written as Structured Text:
```iecst
PROGRAM _CYCLIC
(* Network 1 *)
gCtrl.squaring.frontSquaringEquipped := UDINT_TO_BOOL(gConfigApp.options.frontSquaringOption);

(* Network 2: ===================================================================================== Side Squaring *)
gMachineIO.dout.SideSquaringExtend_SOL8A := gCtrl.main.noFaults AND gCtrl.squaring.hmiBtnSidePlatesExtRet;

(* Network 3 *)
gMachineIO.dout.SideSquaringRetract_SOL8B := NOT gMachineIO.dout.SideSquaringExtend_SOL8A;

(* Network 4: ===================================================================================== Front Squaring *)
gMachineIO.dout.FrontSquaringExtend_SOL11A := gCtrl.main.noFaults AND gCtrl.squaring.hmiBtnFrontPlateExtRet;

(* Network 5 *)
gMachineIO.dout.FrontSquaringRetract_SOL11B := NOT gMachineIO.dout.FrontSquaringExtend_SOL11A;
END_PROGRAM
```

### Program Logical/paiComponents/bglib

#### bgftpclient.c
```c
#include <bur/plc.h>
#include <bur/plctypes.h>
#include <ethsock.h>
#include <astcp.h>
#include <asstring.h>
#include <brsystem.h>
#include <sys_lib.h>

#include "bgsprintf.h"
#include "bgstatemachine.h"
#include "bgstring.h"
#include "bgFtpClient.h"

#include "bgdebug.h"

#include "bgstatemachine.c"
#include "bgsprintf.c"
#include "bgstring.c"

/*
History:
7/22/2007
- updated to a new, AsTcp library

9/11/2005
- added support for receiving large files over ftp
- added error event for user ftp commands:
int bgFtpClientCmd<CmdName>OnError(bgFtpClient_typ *p);

*/

void ftpClientConnect(bgFtpClient_typ *p, int msgId);
int ftpClientConnectOnDone(bgFtpClient_typ *p);
int ftpClientConnectOnError(bgFtpClient_typ *p);

void ftpClientLogin(bgFtpClient_typ *p, int msgId);
int ftpClientLoginOnDone(bgFtpClient_typ *p);
int ftpClientLoginOnError(bgFtpClient_typ *p);

void ftpClientLogout(bgFtpClient_typ *p, int msgId);
int ftpClientLogoutOnDone(bgFtpClient_typ *p);
int ftpClientLogoutOnError(bgFtpClient_typ *p);

void ftpClientCmdGetFile(bgFtpClient_typ *p);

void ftpClientCmdList(bgFtpClient_typ *p);

void ftpClientCmdPwd(bgFtpClient_typ *p);

void ftpClientCmdCwd(bgFtpClient_typ *p);

void ftpClientDataServer(bgFtpClient_typ *p, int msgId);
int ftpClientDataServerOnError(bgFtpClient_typ *p);
int ftpClientDataServerOnDone(bgFtpClient_typ *p);

void ftpClientSingleCmdInit(bgFtpClient_typ *p, char *cmd, char *expectedServerResponse);
void ftpClientSingleCmd(bgFtpClient_typ *p);
int ftpClientSingleCmdOnError(bgFtpClient_typ *p);
int ftpClientSingleCmdOnDone(bgFtpClient_typ *p);

void ftpClientExecuteUserCmd_cyclic(bgFtpClient_typ *p);

int ftpClientCmdMultiOnDone(bgFtpClient_typ *p, int cmdId);
int ftpClientMultiCmdOnError(bgFtpClient_typ *p, int cmdId);
int ftpClientCmdCheckServerResponseCode(bgFtpClient_typ *p);

void ftpClientInitDataPort(bgFtpClient_typ *p);
void swapBytesInShort(unsigned short *value);
void setSocketAddressData(ETH_sockaddr_typ *adrData, char *hostIpAddressString, unsigned short hostPort);
void ftpClientGetResponse(bgFtpClient_typ *p);

void ftpClientCmdTextPort(bgFtpClient_typ *p, char *textBuffer);
void ftpClientMutliStateCmdErrorLog(bgFtpClient_typ *p);

int ftpClientIncrDataPort(bgFtpClient_typ *p);

/*
########################################################################################
========================================================================================
- FTP client protocol main state machine
- must be executed as a cyclic task (<=100ms)
- protocol implemenation uses nested state machines (several levels deep)
- FTP functions such as: connect, disconnect, login, logout and different FTP commands
are all implemented as state machines
*/
void bgFtpClientCyclic(bgFtpClient_typ *p, int msgId)
{
bgStateMachine_typ *psm = &p->smFtp;

	/*FTP client top level state machine*/
	switch( bgSMCyclic(psm) ){
		case 1:
          	/*idle; monitor user connection request flag*/
			bgSMSetStateName(psm, "Idle");

          	if(p->user.connectRequest){
	            p->user.connectRequest = 0;
	            p->user.disconnectRequest = 0;
				bgSMSetNextState(psm, bgSMGetState(psm) + 1);
          	}
		break;
		case 2:
			/*connect to FTP server*/
			bgSMSetStateName(psm, "Connect");

			if(bgSMIsStateInit(psm)){
				ftpClientConnect(p, BGSM_MSGID_INIT);
			}

			ftpClientConnect(p, BGSM_MSGID_CYCLIC);

			/*check if we are connected to FTP server*/
			if( p->isConnected ){
				bgSMSetNextState(psm, bgSMGetState(psm) + 1);
			}

			if(	ftpClientConnectOnError(p)){
                ERRxwarning(USER_ERROR_FTP, 1, "ftpClient-Err-socket()");
				bgSMRaiseError(psm, "error in lower level SM", 1, 0);
            }
		break;
		case 3:
			/*login*/
			bgSMSetStateName(psm, "Login");

			if(bgSMIsStateInit(psm)){
				ftpClientLogin(p, BGSM_MSGID_INIT);
			}

			ftpClientLogin(p, BGSM_MSGID_CYCLIC);

			/*check if we are looged-in*/
			if(p->isLoggedIn){
				p->userState = 0;
				bgSMSetNextState(psm, bgSMGetState(psm) + 1);
			}
			if(ftpClientLoginOnError(p)){
                ERRxwarning(USER_ERROR_FTP, 1, "ftpClient-Err-login()");
				bgSMRaiseError(psm, "error in lower level SM", 0, 0);
            }
		break;
		case 4:
            /*connected & logged-in -> normal operational state*/
			bgSMSetStateName(psm, "Ready");

			/*monitor requests & execute FTP commands*/
			ftpClientExecuteUserCmd_cyclic(p);

			/*terminate if socket error detected*/
			if(p->cmdError == ERR_SOCKET){
				bgSMSetNextState(psm, bgSMGetState(psm) + 1);
			}

			if(p->test){
				p->test = 0;
				ftpClientGetResponse(p);
			}

            /*monitor user disconnect request*/
            /*NOTE: upon receiving request, make sure to wait that FTP command in progress completes!*/

			/*disconnect allowed only after command completes*/
            if(p->user.disconnectRequest && !p->userState){
                p->user.connectRequest = 0;
                p->user.disconnectRequest = 0;
				bgSMSetNextState(psm, bgSMGetState(psm) + 1);
            }
		break;
		case 5:
            /*logout*/
			bgSMSetStateName(psm, "Logout");

			if(bgSMIsStateInit(psm)){
				ftpClientLogout(p, BGSM_MSGID_INIT);
			}

			ftpClientLogout(p, BGSM_MSGID_CYCLIC);

			/*chech if we are logged out*/
			if(!p->isLoggedIn){
				bgSMSetNextState(psm, bgSMGetState(psm) + 1);
			}

			if(ftpClientLogoutOnError(p)){
                ERRxwarning(USER_ERROR_FTP, 1, "ftpClient-Err-socket()");
				bgSMRaiseError(psm, "error in lower level SM", 0, 0);
            }
		break;
		case 6:
			bgSMSetStateName(psm, "Close CMD socket");
            /*normal operation; close socket*/
			bgSMRaiseDone(psm, 0);
		break;
		default:
			/*unhandled state*/
			bgSMRaiseError(psm, "unknown state", 0, bgSMGetState(psm));
		break;
	}

	if(bgSMOnDone(psm)){
		/*error state; socket closing is needed*/
		close(p->sock);

		p->isConnected = 0;

		bgSMSetNextState(psm, 1);
	}

	if(bgSMOnError(psm)){
		/*check if socket close needed or not?*/
		if( !bgSMGetErrorId(psm) )
			close(p->sock);

		p->isConnected = 0;
		p->cmdError = 1;
		bgSMSetNextState(psm, 1);
	}
}
/*
########################################################################################
	 INDIVIDUAL FTP COMMANDS
- each individual FTP command has following USER level interface methods:
	ftpClientCmd<Name>Init()
		- start command execution; pass-in user parameters; init cmd state machine
	ftpClientCmd<Name>OnDone()
		- monitor cmd completion (0-not complete; 1-complete)

- each command also has core implemenation (not used or called by the user)
	ftpClientCmd<Name>()

- FTP commands such as: PWD, CWD, PUT, GET, DIR are multi-level commands: it usually takes
several primitive FTP commands (i.e. PORT, TYPE, RETR etc) to complete one FTP command

########################################################################################
*/

/*
========================================================================================
- state machine that handles execution of individual, multi-level FTP commands
- FTP client executes one Multi-level command at the time
*/
void ftpClientExecuteUserCmd_cyclic(bgFtpClient_typ *p)
{
	/*execute user commands*/
	switch(p->userState){
	/*idle*/
        case 0:
        break;
        case 1:
        break;
        case 2:
            ftpClientCmdList(p);
        break;
        case 4:
            ftpClientCmdPwd(p);
        break;
        case 6:
            ftpClientCmdGetFile(p);
        break;
        case 8:
            ftpClientCmdCwd(p);
        break;
        default:
            p->userState = 0;
        break;
	}

}

/*
========================================================================================
FTP Command Implementation:
GetFile
*/
void bgFtpClientCmdGetFileInit(bgFtpClient_typ *p, char *fileName, char* buffer, int bufferLength)
{
    /*select command to execute*/
	p->userState = 6;

	/*pass command parameters*/
	p->user.dataBuffer = buffer;
	p->user.dataBufferLength = bufferLength;
	brsstrcpy((UDINT)&p->user.fileName[0], (UDINT)fileName);

    /*start command execution*/
	bgSMReset(&p->smFtpMultiCmd);
}

int bgFtpClientCmdGetFileOnDone(bgFtpClient_typ *p)
{
	return ftpClientCmdMultiOnDone(p, 6);
}

int bgFtpClientCmdGetFileOnError(bgFtpClient_typ *p)
{
	return ftpClientMultiCmdOnError(p, 6);
}

void ftpClientCmdGetFile(bgFtpClient_typ *p)
{
char cmdText[256];
bgStateMachine_typ *psm = &p->smFtpMultiCmd;

	/*FTP client multi level command state machine*/
	switch( bgSMCyclic(psm) ){
		case 1:
          	/*idle - monitor user connection request flag*/
			bgSMSetStateName(psm, "GetFile-InitDataSocket");

			if( bgSMIsStateInit(psm) ){
				/*generate port number to use*/
				ftpClientIncrDataPort(p);
				/*init Data transport socket*/
	            ftpClientDataServer(p, BGSM_MSGID_INIT);
			}

			/*wait for ready msg from the DataServer*/
            if( p->isDataPortReady ){
				bgSMSetNextState(psm, bgSMGetState(psm) + 1);
            }
/*TODO: timeout*/
		break;
		case 2:
    		/*PORT command: "PORT 192,168,1,6,0,20<CR><LF>"*/
			bgSMSetStateName(psm, "GetFile-PORT");
			if(bgSMIsStateInit(psm)){
	    		/*send command*/
	            ftpClientCmdTextPort(p, &cmdText[0]);

	    		ftpClientSingleCmdInit(p, &cmdText[0], "2??");
			}

    		/*recv cmd response*/
    		ftpClientSingleCmd(p);
			if(ftpClientSingleCmdOnDone(p)){
				bgSMSetNextState(psm, bgSMGetState(psm) + 1);
			}
			if(ftpClientSingleCmdOnError(p)){
				bgSMRaiseError(psm, "error in lower level SM", 0, 0);
			}
		break;
		case 3:
    		/*TYPE command: "TYPE I<CR><LF>"*/
			bgSMSetStateName(psm, "GetFile-TYPE");
			if(bgSMIsStateInit(psm)){
	    		/*send command*/
	    		ftpClientSingleCmdInit(p, "TYPE I", "2??");
			}

    		/*recv cmd response*/
    		ftpClientSingleCmd(p);
			if(ftpClientSingleCmdOnDone(p)){
				bgSMSetNextState(psm, bgSMGetState(psm) + 1);
			}

			if(ftpClientSingleCmdOnError(p)){
				bgSMRaiseError(psm, "error in lower level SM", 0, 0);
			}
		break;
		case 4:
    		/*RETR command: "RETR<CR><LF>""*/
			bgSMSetStateName(psm, "GetFile-RETR");
			if(bgSMIsStateInit(psm)){
	    		/*send command*/
	    		/*send command*/
	    		brsstrcpy((UDINT)&cmdText[0], (UDINT)"RETR ");
	    		brsstrcat((UDINT)&cmdText[0], (UDINT)&p->user.fileName[0]);
	    		ftpClientSingleCmdInit(p, &cmdText[0], "2??");
			}

    		/*recv cmd response*/
    		ftpClientSingleCmd(p);
			if(ftpClientSingleCmdOnDone(p)){
				/*notify data port server that the response is comming*/
				ftpClientDataServer(p, 2);
				bgSMSetNextState(psm, bgSMGetState(psm) + 1);
			}

			if(ftpClientSingleCmdOnError(p)){
				bgSMRaiseError(psm, "error in lower level SM", 0, 0);
				/*close data server port*/
				ftpClientDataServer(p, 3);
			}
		break;
        case 5:
			bgSMSetStateName(psm, "GetFile-DATASRVR active");
        break;
		default:
			/*unhandled state*/
			bgSMRaiseError(psm, "unknown state", 0, bgSMGetState(psm));
		break;
	}

	if(bgSMOnError(psm)){
		p->isErrorMultiCmd = p->userState;
		p->userState = 0;
		return;
	}

	ftpClientDataServer(p, BGSM_MSGID_CYCLIC);

	if(ftpClientDataServerOnDone(p)){
		p->isDoneMultiCmd = p->userState;
		p->userState = 0;
	}

	if(ftpClientDataServerOnError(p)){
		p->isErrorMultiCmd = p->userState;
		p->userState = 0;
	}

}
/*
========================================================================================
FTP Command Implementation:
List (dir)
*/
void bgFtpClientCmdListInit(bgFtpClient_typ *p, char *buffer, int bufferLength)
{
    /*select command to execute*/
	p->userState = 2;

	/*pass command parameters*/
	p->user.dataBuffer = buffer;
	p->user.dataBufferLength = bufferLength;

    /*start command execution*/
	bgSMReset(&p->smFtpMultiCmd);
}

int bgFtpClientCmdListOnDone(bgFtpClient_typ *p)
{
	return ftpClientCmdMultiOnDone(p, 2);
}

int bgFtpClientCmdListOnError(bgFtpClient_typ *p)
{
	return ftpClientMultiCmdOnError(p, 2);

}

void ftpClientCmdList(bgFtpClient_typ *p)
{
char cmdText[64];
bgStateMachine_typ *psm = &p->smFtpMultiCmd;

	/*FTP client multi level command state machine*/
	switch( bgSMCyclic(psm) ){
		case 1:
          	/*idle - monitor user connection request flag*/
			bgSMSetStateName(psm, "List-InitDataSocket");

			if( bgSMIsStateInit(psm) ){
				/*generate port number to use*/
				ftpClientIncrDataPort(p);
				/*init Data transport socket*/
	            ftpClientDataServer(p, BGSM_MSGID_INIT);
			}

			/*wait for ready msg from the DataServer*/
            if( p->isDataPortReady ){
				bgSMSetNextState(psm, bgSMGetState(psm) + 1);
            }
/*TODO: timeout*/
		break;
		case 2:
    		/*PORT command: "PORT 192,168,1,6,0,20<CR><LF>"*/
			bgSMSetStateName(psm, "List-PORT");
			if(bgSMIsStateInit(psm)){
	    		/*send command*/
	            ftpClientCmdTextPort(p, &cmdText[0]);

	    		ftpClientSingleCmdInit(p, &cmdText[0], "2??");
			}

    		/*recv cmd response*/
    		ftpClientSingleCmd(p);
			if(ftpClientSingleCmdOnDone(p)){
				bgSMSetNextState(psm, bgSMGetState(psm) + 1);
			}
			if(ftpClientSingleCmdOnError(p)){
				bgSMRaiseError(psm, "error in lower level SM", 0, 0);
			}
		break;
		case 3:
    		/*TYPE command: "TYPE I<CR><LF>"*/
			bgSMSetStateName(psm, "List-TYPE");
			if(bgSMIsStateInit(psm)){
	    		/*send command*/
	    		ftpClientSingleCmdInit(p, "TYPE I", "2??");
			}

    		/*recv cmd response*/
    		ftpClientSingleCmd(p);
			if(ftpClientSingleCmdOnDone(p)){
				bgSMSetNextState(psm, bgSMGetState(psm) + 1);
			}

			if(ftpClientSingleCmdOnError(p)){
				bgSMRaiseError(psm, "error in lower level SM", 0, 0);
			}
		break;
		case 4:
    		/*LIST command: "LIST<CR><LF>""*/
			bgSMSetStateName(psm, "List-List");
			if(bgSMIsStateInit(psm)){
	    		/*send command*/
	    		ftpClientSingleCmdInit(p, "LIST", "2??");
			}

    		/*recv cmd response*/
    		ftpClientSingleCmd(p);
			if(ftpClientSingleCmdOnDone(p)){
				/*notify data port server that the response is comming*/
				ftpClientDataServer(p, 2);
				bgSMSetNextState(psm, bgSMGetState(psm) + 1);
			}

			if(ftpClientSingleCmdOnError(p)){
				/*close data server port*/
				ftpClientDataServer(p, 3);
				bgSMRaiseError(psm, "error in lower level SM", 0, 0);
			}
		break;
        case 5:
			bgSMSetStateName(psm, "List-DATASRVR active");
        break;
		default:
			/*unhandled state*/
			bgSMRaiseError(psm, "unknown state", 0, bgSMGetState(psm));
		break;
	}

	if(bgSMOnError(psm)){
		p->isErrorMultiCmd = p->userState;
		p->userState = 0;
		return;
	}

	ftpClientDataServer(p, BGSM_MSGID_CYCLIC);

	if(ftpClientDataServerOnDone(p)){
		p->isDoneMultiCmd = p->userState;
		p->userState = 0;
	}

	if(ftpClientDataServerOnError(p)){
		p->isErrorMultiCmd = p->userState;
		p->userState = 0;
	}
}
/*
========================================================================================
FTP Command Implementation:
Pwd (Print Working Directory)
*/
void bgFtpClientCmdPwdInit(bgFtpClient_typ *p, char *buffer, int bufferLength)
{
    /*select command to execute*/
	p->userState = 4;

	/*pass command parameters*/
	p->user.dataBuffer = buffer;
	p->user.dataBufferLength = bufferLength;

    /*start command execution*/
	bgSMReset(&p->smFtpMultiCmd);
}

int bgFtpClientCmdPwdOnDone(bgFtpClient_typ *p)
{
	return ftpClientCmdMultiOnDone(p, 4);
}

int bgFtpClientCmdPwdOnError(bgFtpClient_typ *p)
{
	return ftpClientMultiCmdOnError(p, 4);

}

void ftpClientCmdPwd(bgFtpClient_typ *p)
{
bgStateMachine_typ *psm = &p->smFtpMultiCmd;

	/*FTP client multi level command state machine*/
	switch( bgSMCyclic(psm) ){
		case 1:
    		/*XPWD command: "XPWD<CR><LF>"*/
			bgSMSetStateName(psm, "PWD");
			if(bgSMIsStateInit(psm)){
	    		/*send command*/
	    		ftpClientSingleCmdInit(p, "PWD", "2??");
			}

    		/*recv cmd response*/
    		ftpClientSingleCmd(p);

			if(ftpClientSingleCmdOnDone(p)){
				/*copy response strig into the user supplied buffer*/
				brsstrcpy((UDINT)p->user.dataBuffer, (UDINT)p->responseList.items[0]);
				bgSMRaiseDone(psm, 0);
			}

			if(ftpClientSingleCmdOnError(p)){
				bgSMRaiseError(psm, "got lower SM error", 0, 0);
			}
		break;
		default:
			/*unhandled state*/
			bgSMRaiseError(psm, "unknown state", 0, bgSMGetState(psm));
		break;
	}

	if(bgSMOnError(psm)){
		p->userState = 0;
	}

	if(bgSMOnDone(psm)){
		p->isDoneMultiCmd = p->userState;
		p->userState = 0;
	}

}
/*
========================================================================================
FTP Command Implementation:
Cwd (Change Working Directory)
*/
void bgFtpClientCmdCwdInit(bgFtpClient_typ *p, char *fileName, char *buffer, int bufferLength)
{
    /*select command to execute*/
	p->userState = 8;

	/*pass command parameters*/
	p->user.dataBuffer = buffer;
	p->user.dataBufferLength = bufferLength;
	brsstrcpy((UDINT)&p->user.fileName[0], (UDINT)fileName);

    /*start command execution*/
	bgSMReset(&p->smFtpMultiCmd);

}

int bgFtpClientCmdCwdOnDone(bgFtpClient_typ *p)
{
	return ftpClientCmdMultiOnDone(p, 8);
}

int bgFtpClientCmdCwdOnError(bgFtpClient_typ *p)
{
	return ftpClientMultiCmdOnError(p, 8);

}

void ftpClientCmdCwd(bgFtpClient_typ *p)
{
char cmdText[255];

bgStateMachine_typ *psm = &p->smFtpMultiCmd;

	/*FTP client multi level command state machine*/
	switch( bgSMCyclic(psm) ){
		case 1:
    		/*XPWD command: "CWD <fileName><CR><LF>"*/
			bgSMSetStateName(psm, "CWD");
			if(bgSMIsStateInit(psm)){
	    		/*send command: "CWD <fileName><CR><LF>"*/
	    		brsstrcpy((UDINT)&cmdText[0], (UDINT)"CWD ");
	    		brsstrcat((UDINT)&cmdText[0], (UDINT)&p->user.fileName[0]);
	    		ftpClientSingleCmdInit(p, &cmdText[0], "2??");
			}

    		/*recv cmd response*/
    		ftpClientSingleCmd(p);

			if(ftpClientSingleCmdOnDone(p)){
				/*copy response strig into the user supplied buffer*/
				brsstrcpy((UDINT)p->user.dataBuffer, (UDINT)p->responseList.items[0]);
				bgSMRaiseDone(psm, 0);
			}

			if(ftpClientSingleCmdOnError(p)){
				bgSMRaiseError(psm, "got lower SM error", 0, 0);
			}
		break;
	}

	if(bgSMOnError(psm)){
		p->isErrorMultiCmd = p->userState;
		p->userState = 0;
		return;
	}

	if(bgSMOnDone(psm)){
		p->isDoneMultiCmd = p->userState;
		p->userState = 0;
	}
}
/*
########################################################################################
========================================================================================
FTP Connect command state machine:
*/
int ftpClientConnectOnDone(bgFtpClient_typ *p){
	return bgSMOnDone(&p->smCmdSocket);
}

int ftpClientConnectOnError(bgFtpClient_typ *p){
	return bgSMOnError(&p->smCmdSocket);
}

void ftpClientConnect(bgFtpClient_typ *p, int msgId)
{
DINT ret;
bgStateMachine_typ *psm = & p->smCmdSocket;

	if( msgId == BGSM_MSGID_INIT){
		bgSMReset(psm);
	}

    switch(bgSMCyclic(psm)){
        case 1:
			bgSMSetStateName(psm, "Connect-CreateSocket");

			if( bgSMIsStateInit(psm) ){
				p->cmdError = 0;
				p->cmdErrorCode = 0;
				p->isConnected = 0;
				/*create socket*/
				p->sock = socket(ETH_AF_INET, ETH_SOCK_STREAM, 0);

				if( p->sock == ERR_SOCKET ){
					bgSMRaiseError(psm, "socket create err", 0, EthGetError());
					break;
				}

				/*set non-blocking socket operation*/
				{
					UDINT arg = 1;
					ioctl(p->sock, ETH_FIONBIO, (UDINT)&arg);
				}

				/*reset select flags*/
				fd_zero((UDINT)&p->fdR);
				fd_zero((UDINT)&p->fdW);

				/*set time-out to 10ms*/
				p->timeOut.tv_sec = 0;
				p->timeOut.tv_usec = 1000 * 10;

				/*adjust my own timeout counters*/
				p->sockData_TimerCounter = 0;
				p->sockData_TimerTime = 10;
#if 0
/*bind not necessary*/
				/*bind client socket*/
				ret = bind(p->sock, (UDINT)&p->ftpClientAdrData, sizeof(p->ftpClientAdrData));
				if(ret == ERR_SOCKET){
					bgSMRaiseError(psm, "socket bind err", 0, EthGetError());
					break;
				}
#endif
			}

			/*connect to remote host*/
			ret = connect(p->sock, (UDINT)&p->ftpServerAdrCmd, sizeof(p->ftpServerAdrCmd) );

			if(ret == ERR_SOCKET){
				UINT errCode = EthGetError();
				if(errCode == ERR_ETH_INPROGRESS){
					/*next: wait connect to complete*/
					bgSMSetNextState(psm, bgSMGetState(psm) + 1);
				    break;
				}else
				if(errCode == ERR_ETH_ISCONN){
					/*it's connected -> done*/
					ERRxwarning(USER_ERROR_FTP, errCode, "connect()-alreadyOK!");
					bgSMRaiseDone(psm, 0);
					break;
				}
				else{
					bgSMRaiseError(psm, "socket connect err", 0, EthGetError());
					break;
				}
			}
			/*connected!*/
			ERRxwarning(USER_ERROR_FTP, ret, "connect()-OK-Quick!");
			bgSMRaiseDone(psm, 0);
		break;
		case 2:
			bgSMSetStateName(psm, "Connect-Connect");

			/*select waits for connection to complete*/
			fd_set(p->sock, (UDINT)&p->fdR);
			fd_set(p->sock, (UDINT)&p->fdW);
			ret = sock_select(32, (UDINT)&p->fdR, (UDINT)&p->fdW, 0L, (UDINT)&p->timeOut);

			if(ret == ERR_SOCKET){
				bgSMRaiseError(psm, "socket connect err", 0, EthGetError());
				break;
			}
/*
			DBG("connect: ret=%d, error=%d\n\r", ret, EthGetError());
*/
			if(ret == 0){
				if( p->sockData_TimerCounter >= p->sockData_TimerTime ){
					/*NOTES:
					- trying to figure out how does the select timeout works in B&R!
					- using EthGetError() here is not needed, just to see what comes back
					*/
					bgSMRaiseError(psm, "connect timeout", 0, EthGetError());
				}else{
					p->sockData_TimerCounter++;
				}
			}else{
				if( fd_isset(p->sock, (UDINT)&p->fdW) ){
					bgSMRaiseDone(psm, 0);
				}
			}
		break;
		default:
			/*unhandled state*/
			bgSMRaiseError(psm, "unknown state", 0, bgSMGetState(psm));
		break;
    }

	if( bgSMOnDone(psm)){
		ERRxwarning(USER_ERROR_FTP, 0, "connect()-OK!");
		p->isConnected = 1;
	}

	if( bgSMOnError(psm)){

	}
}
/*
========================================================================================
*/
void ftpClientMutliStateCmdErrorLog(bgFtpClient_typ *p){
char text[64];
	/*log error*/
	brsstrcpy((UDINT)&text[0], (UDINT)"Err: ");
	brsstrcat((UDINT)&text[0], (UDINT)&p->cmdSendBuf[0]);
    ERRxwarning(USER_ERROR_FTP, p->cmdErrorCode, &text[0]);
}
/*
########################################################################################
========================================================================================
FTP Login command state machine:
-return values:
*/
int ftpClientLoginOnDone(bgFtpClient_typ *p){
	return bgSMOnDone(&p->smFtpMultiCmd);
}

int ftpClientLoginOnError(bgFtpClient_typ *p){
	return bgSMOnError(&p->smFtpMultiCmd);
}
void ftpClientLogin(bgFtpClient_typ *p, int msgId)
{
bgStateMachine_typ *psm = &p->smFtpMultiCmd;

	if( msgId == BGSM_MSGID_INIT){
		bgSMReset(psm);
	}

    switch(bgSMCyclic(psm)){
        case 1:
			/*send USER name*/
			bgSMSetStateName(psm, "Login-Welcome");

			if( bgSMIsStateInit(psm) ){
				/*send request*/
				/*ftpClientSingleCmdInit(p, 0, ">name");*/
				ftpClientSingleCmdInit(p, 0, ">FTP");
			}

			/*recv response*/
			ftpClientSingleCmd(p);

			if(ftpClientSingleCmdOnDone(p)){
				bgSMSetNextState(psm, bgSMGetState(psm) + 1);
			}

			if(ftpClientSingleCmdOnError(p)){
				bgSMRaiseError(psm, "error in lower level SM", 0, 0);
			}
        break;
        case 2:
			/*send USER name*/
			bgSMSetStateName(psm, "Login-UserName");

			if( bgSMIsStateInit(psm) ){
				/*send request*/
				ftpClientSingleCmdInit(p, "USER  anonymous", "331");
			}

			/*recv response*/
			ftpClientSingleCmd(p);

			if(ftpClientSingleCmdOnDone(p)){
				bgSMSetNextState(psm, bgSMGetState(psm) + 1);
			}

			if(ftpClientSingleCmdOnError(p)){
				bgSMRaiseError(psm, "error in lower level SM", 0, 0);
			}
        break;
        case 3:
			/*send PASSWORD */
			bgSMSetStateName(psm, "Login-Password");

			if( bgSMIsStateInit(psm) ){
				/*send request*/
				ftpClientSingleCmdInit(p, "PASS  anonymous@", "230");
			}

			/*recv response*/
			ftpClientSingleCmd(p);

			if(ftpClientSingleCmdOnDone(p)){
				bgSMRaiseDone(psm, 0);
			}

			if(ftpClientSingleCmdOnError(p)){
				bgSMRaiseError(psm, "error in lower level SM", 0, 0);
			}
        break;
        default:
			/*unhandled state*/
			bgSMRaiseError(psm, "unknown state", 0, bgSMGetState(psm));
        break;
    }

	if( bgSMOnDone(psm) ){
		p->isLoggedIn = 1;
	}

	if( bgSMOnError(psm) ){
		ftpClientMutliStateCmdErrorLog(p);
	}

}
/*
########################################################################################
========================================================================================
FTP Logout command state machine:
-return values:
*/
int ftpClientLogoutOnDone(bgFtpClient_typ *p){
	return bgSMOnDone(&p->smFtpMultiCmd);
}

int ftpClientLogoutOnError(bgFtpClient_typ *p){
	return bgSMOnError(&p->smFtpMultiCmd);
}

void ftpClientLogout(bgFtpClient_typ *p, int msgId)
{
bgStateMachine_typ *psm = &p->smFtpMultiCmd;

	if( msgId == BGSM_MSGID_INIT){
		bgSMReset(psm);
	}

    switch(bgSMCyclic(psm)){
        case 1:
			/*send USER name*/
			bgSMSetStateName(psm, "Logout-Quit");

			if( bgSMIsStateInit(psm) ){
				/*send request*/
				ftpClientSingleCmdInit(p, "QUIT", "2??");
			}

			/*recv response*/
			ftpClientSingleCmd(p);

			if(ftpClientSingleCmdOnDone(p)){
				bgSMRaiseDone(psm, 0);
			}

			if(ftpClientSingleCmdOnError(p)){
				bgSMRaiseError(psm, "error in lower level SM", 0, 0);
			}
        break;
        default:
			/*unhandled state*/
			bgSMRaiseError(psm, "unknown state", 0, bgSMGetState(psm));
        break;
    }

	if(bgSMOnDone(psm)){
		p->isLoggedIn = 0;
	}

	if(bgSMOnError(psm)){
		p->isLoggedIn = 0;
		ftpClientMutliStateCmdErrorLog(p);
	}
}
/*
########################################################################################
========================================================================================
Lowest level state machine handles execution of a single FTP request/response messaging

ftpClientSingleCmdInit();
	- selects command to execute; init command state machine

ftpClientSingleCmd();
	- command execution state machine

ftpClientCmdCheckServerResponseCode()
	- command response check and verification

*/
void ftpClientSingleCmdInit(bgFtpClient_typ *p, char *cmd, char *expectedServerResponse){
int i;

	/*copy command string into send buffer*/
	p->cmdSendBuf[0]=0;
	if(cmd){
		brsstrcpy((UDINT)&p->cmdSendBuf[0], (UDINT)cmd);
		/*append string termination -> CRLF*/
		brsstrcat((UDINT)&p->cmdSendBuf[0], (UDINT)"\r\n");
	}

	/*define expected server response string?*/
	p->cmdExpectedServerResponse[0] = 0;	/*don't care*/
	if(expectedServerResponse){
		/*is expected server response code or string?*/
		if( *expectedServerResponse == '>'){
			i = 1;
			p->cmdExpectedServerResponseCodeOrString = 1;	/*string*/
		}else{
			i = 0;
			p->cmdExpectedServerResponseCodeOrString = 0;	/*code*/
		}
		bgStrCpyN(&p->cmdExpectedServerResponse[0], expectedServerResponse+i, FTPCLIENT_RESPONSECODE_LEN);
	}

	/*clr rcv buffer string*/
	memset(&p->cmdRecvBuf[0], 0, FTPCLIENT_CMDBUFSIZE);
#if 0
/*clear response lines*/
	/*init ptrs*/
	p->responseList.maxCount = CMD_RESPONSE_MAXLINES;
	p->responseList.lines[0] = &p->responseList.line0[0];
	p->responseList.lines[1] = &p->responseList.line1[0];
	p->responseList.lines[2] = &p->responseList.line2[0];
	p->responseList.lines[3] = &p->responseList.line3[0];
	p->responseList.lines[4] = &p->responseList.line4[0];

	/*clear all response lines*/
	for(i=0;i<CMD_RESPONSE_MAXLINES; i++){
		memset(p->responseList.lines[i], 0, CMD_RESPONSE_MAXLINELEN);
	}
	/*number of lines retrieved from the cmd buffer*/
	p->responseList.count = 0;
#endif
	/*number of lines retrieved from the cmd buffer*/
	p->responseList.itemCount = 0;

	/*reset command execution state machine*/
	bgSMReset(&p->smFtpCmd);
}

void ftpClientSingleCmd(bgFtpClient_typ *p){
DINT len;
DINT ret;
bgStateMachine_typ *psm = &p->smFtpCmd;

	/*state machine states*/
	switch( bgSMCyclic(psm) ){
		case 1:
          	/*send command request*/
			bgSMSetStateName(psm, "ftpSingleCmd");

			if(bgSMIsStateInit(psm)){
				/*check input conditions and paramters*/
				if( !p->isConnected ){
					bgSMRaiseError(psm, "not connected", 0, 0);
					break;
				}
				if( !p->cmdSendBuf[0]){
					/*nothing to send! receive only (i.e. welcome message just after connect()*/
					break;
				}

				/*send command to server*/
	         	len = strlen(&p->cmdSendBuf[0]);
	        	ret = send(p->sock, (UDINT)&p->cmdSendBuf[0], len, 0L);

	        	if(ret == ERR_SOCKET){
					bgSMRaiseError(psm, "send() error", 0, EthGetError());
					break;
	        	}

				/*remember the send length*/
				DBG("Single CMD send();Bytes=%d;[%s]\r\n", (int)ret, &p->cmdSendBuf[0]);
				p->sendLen = ret;
				return;
			}

	       	/*call receive (NON BLOCKING MODE!)*/
        	ret = recv(p->sock, (UDINT)&p->cmdRecvBuf[0],  FTPCLIENT_CMDBUFSIZE, 0L);

        	if(ret == ERR_SOCKET){
        		UINT errCode = EthGetError();
        		/*none blocking receive return this following value if data is not available yet*/
        		if( errCode == ERR_ETH_WOULDBLOCK ){
        			/*wait response*/
					return;
        		}

				/*recv error*/
				bgSMRaiseError(psm, "recv() error", 0, EthGetError());
				break;
        	}

			if(ret == 0){
				bgSMRaiseError(psm, "rx len=0", 0, 0);
				return;
			}

			/*receive is complete; store receive length & terminate rx buffer*/
			p->cmdRecvBuf[ret] = 0;
			DBG("Single CMD recv();Bytes=%d;[%s]\r\n", (int)ret, &p->cmdRecvBuf[0]);
			p->recvLen = ret;

			ret = ftpClientCmdCheckServerResponseCode(p);

			if( ret == 1)
				bgSMRaiseDone(psm, 0);

			if( ret == 2)
				bgSMRaiseError(psm, "server error response", 0, 0);

		break;
		default:
			/*unhandled state*/
			bgSMRaiseError(psm, "unknown state", 0, bgSMGetState(psm));
		break;
	}

	/*error event handler*/
	if(bgSMOnError(psm)){
		DBG("ftpClientSingleCmd - ERROR.\r\n");
	}

	/*done event handler*/
	if(bgSMOnDone(psm)){
		DBG("ftpClientSingleCmd - DONE.\r\n");
	}
}

int ftpClientSingleCmdOnError(bgFtpClient_typ *p)
{
	return bgSMOnError(&p->smFtpCmd);
}

int ftpClientSingleCmdOnDone(bgFtpClient_typ *p)
{
	return bgSMOnDone(&p->smFtpCmd);
}

/*
========================================================================================
FTP command response code is an ASCII line that looks like:
"xyz-response text<CR><LF>"
where x,y,z are numeric chars <0-9> followed by a '-' and the response text
- multiple lines per response are possible
- this function retrieves the response from the server, formats it into a list (array) of lines
and then searches each line for the user supplied code (res1,res2,res3)
- if res<x> is given as 0, it means don't care (see ftp spec)

*/
int ftpClientCmdCheckServerResponseCode(bgFtpClient_typ *p)
{
char serverResponseCode[3];
char *line;
int result;
int i;

	/*get server's response
	IMPORTANT:
	- note that data for ftpClientGetResponse() method is initilized within ftpClientSingleCmdInit()!
	- order of execution is like:
		init:
			ftpClientSingleCmdInit();
		cyclic:
			if( ftpClientSingleCmd() == DONE )
				if( ftpClientCmdCheckServerResponseCode() == OK )
					nextState;

	- therfore, the ftpClientGetResponse() shall be designed to operate in an incremenal mode: every time
	ftpClientSingleCmd() completes (data is available in the receive buffer) we should just add to the existing lines
	and not delete what we've received till that moment
	*/
	ftpClientGetResponse(p);

	/*final result of the ftpClientCmdCheckServerResponseCode() method:
	0 - response not found (not available -> wait)
	1 - response found (and it's ok; match with expected response)
	2 - response found (and it's not ok; error response from server)
	*/
	p->serverResponseCode = 0;

	/*anything to process!?*/
	if(!p->responseList.itemCount)
		return 0;

	/*check all received response lines every time (not necessary but it's easy to implement and it does not metter*/
	for(i=0; i<p->responseList.itemCount; i++){
		line = p->responseList.items[i];

		if(!p->cmdExpectedServerResponseCodeOrString){
			serverResponseCode[0]=*(line+0);
			serverResponseCode[1]=*(line+1);
			serverResponseCode[2]=*(line+2);

			result = 0;
			if( p->cmdExpectedServerResponse[0] != '?'){
				if(p->cmdExpectedServerResponse[0] == serverResponseCode[0])
					result++;
			}else
				result++;

			if( p->cmdExpectedServerResponse[1] != '?'){
				if(p->cmdExpectedServerResponse[1] == serverResponseCode[1])
					result++;
			}else
				result++;

			if( p->cmdExpectedServerResponse[2] != '?'){
				if(p->cmdExpectedServerResponse[2] == serverResponseCode[2])
					result++;
			}else
				result++;

			if( result >= 3)
				return 1;

			if( (serverResponseCode[0] == '4') || (serverResponseCode[0] == '5'))
				return 2;
		}else{
			result = bgStrFind(line, &p->cmdExpectedServerResponse[0], -1, -1);

			if(result >= 0)
				return 1;
		}
	}

	return 0;
}
/*
========================================================================================
*/
void ftpClientGetResponse(bgFtpClient_typ *p){
int i;
char *src;

	/*ptr to rcv buffer*/
	src = &p->cmdRecvBuf[0];
	p->responseList.src = src;
	bgStringListLines(&p->responseList);

	DBG("Received Cmd Response: lines=%d\r\n", p->responseList.itemCount);
	for(i=0;i<p->responseList.itemCount;i++){
		DBG("Line[%d]=%s\r\n", i, p->responseList.items[i]);
	}

}

int readline(char *src, char *dest, int maxLength){
/*
return: >= 0 (length of the line including CRLF)
return: -1 (no line read)
*/
int lineLen;
char *cPtr;

	lineLen = 0;
	cPtr = src;
	while(maxLength--){

		if( (*cPtr == 0x0D) || ( *cPtr == 0x0A) ){

			lineLen++;
			cPtr++;

			if( (*cPtr == 0x0D) || ( *cPtr == 0x0A) ){
				lineLen++;
			}

			memcpy(dest, src, lineLen);
			*(dest+lineLen+1)= 0;
			return lineLen;
		}

		if( *cPtr == 0 )
			return -1;

		lineLen++;
		cPtr++;
	}

	return -1;
}

/*
========================================================================================
*/
int ftpClientCmdMultiOnDone(bgFtpClient_typ *p, int cmdId)
{
/*generate CmdIsDone signal (1 shoot)*/
	if( p->isDoneMultiCmd == cmdId ){
		p->isDoneMultiCmd = 0;
		return 1;
	}else
		return 0;
}

int ftpClientMultiCmdOnError(bgFtpClient_typ *p, int cmdId){
/*generate CmdIsError signal (1 shoot)*/
	if( p->isErrorMultiCmd == cmdId ){
		p->isErrorMultiCmd = 0;
		return 1;
	}else
		return 0;
}

/*
========================================================================================
*/
void bgFtpClientConnectAndLogin(bgFtpClient_typ *p, char *ethernetDevice, char *serverIp)
{
unsigned long ipAddrClient;

    /*set server ip address and ports to use*/
    /*  21 - standard FTP command port
        20 - standard FTP data port
    */
	setSocketAddressData(&p->ftpServerAdrCmd, serverIp, 21);
	setSocketAddressData(&p->ftpClientAdrData, "", ETH_INADDR_ANY);

	/*retrieve own ip address*/
	p->CfgIPAddr_1.enable = 1;
	p->CfgIPAddr_1.pDevice = (UDINT)ethernetDevice;
	p->CfgIPAddr_1.pIPAddr = (UDINT)&p->CfgIPAddrString[0];
	p->CfgIPAddr_1.Len = 16;
	CfgGetIPAddr(&p->CfgIPAddr_1);

	ipAddrClient = inet_addr( (unsigned long) &p->CfgIPAddrString[0]);

	/*store ip address in an easy format for later use; see PORT command*/
	p->ipAddr[3]= (ipAddrClient>>24)&0xFF;
	p->ipAddr[2]= (ipAddrClient>>16)&0xFF;
	p->ipAddr[1]= (ipAddrClient>>8)&0xFF;
	p->ipAddr[0]= (ipAddrClient)&0xFF;

	p->cmdError = 0;
	p->cmdErrorCode = 0;
	p->isConnected = 0;
    p->user.connectRequest = 1;
}
/*
========================================================================================
*/
int bgFtpClientIsLoggedIn(bgFtpClient_typ *p)
{
    return p->isLoggedIn;
}

/*
========================================================================================
*/
void bgFtpClientDisconnect(bgFtpClient_typ *p)
{
    p->user.disconnectRequest = 1;
}
/*
========================================================================================
*/
int bgFtpClientIsConnected(bgFtpClient_typ *p)
{
    return p->isConnected;
}
/*
========================================================================================
*/
int bgFtpClientIsError(bgFtpClient_typ *p)
{
    return p->cmdError;
}

int ftpClientIncrDataPort(bgFtpClient_typ *p){

	if( !p->dataPort){
		p->dataPort = 190;
	}

	if(p->dataPort>=190)
		p->dataPort++;

	if(p->dataPort>=200)
		p->dataPort = 190;

	return p->dataPort;
}
/*
========================================================================================
*/
void ftpClientCmdTextPort(bgFtpClient_typ *p, char *textBuffer)
{
/*
	bgsprintf(textBuffer, "PORT 192,168,1,6,4,%d", p->dataPort);
*/
	bgsprintf(textBuffer, "PORT %d,%d,%d,%d,4,%d", p->ipAddr[0], p->ipAddr[1], p->ipAddr[2], p->ipAddr[3], p->dataPort);
}
/*
========================================================================================
*/
int ftpClientDataServerOnError(bgFtpClient_typ *p)
{
	return bgSMOnError(&p->smDataSocket);
}

int ftpClientDataServerOnDone(bgFtpClient_typ *p)
{
	return bgSMOnDone(&p->smDataSocket);
}

void ftpClientDataServer(bgFtpClient_typ *p, int msgId)
{
bgStateMachine_typ *psm = &p->smDataSocket;

    /*init data socket (listen)*/
	if( (msgId == BGSM_MSGID_INIT) ){
		bgSMReset(psm);
		p->sockData_TimerTime = 5;
		p->sockData_TimerCounter = 0;
		p->recvLenData = 0;
		p->sendLenData = 0;
		return;
	}

    /*close data socket (listen stop)*/
	if( msgId == 2){
		/*command socket is telling us to receive data from server
		after this event, keep receiving until we don't get any data
		for a certain period of time or the remote host closes the
		connection
		*/
		p->sockData_Timer = 1;
		p->sockData_TimerTime = 10;
		p->sockData_TimerCounter = 0;
		return;
	}

    /*close data socket now!*/
	if( msgId == 3){
		/*command socket is telling us to immediately close data socket
		*/
		bgSMSetNextState(psm, 3);
		return;
	}

	switch(bgSMCyclic(psm)){
		case 1:
			bgSMSetStateName(psm, "DataPort-Open");
			if(bgSMIsStateInit(psm)){

				p->TCPopen_1.enable = 1;
				p->TCPopen_1.port = 4*256 + p->dataPort;
				p->TCPopen_1.pIfAddr = 0;
				p->TCPopen_1.options = 0;
				DBG("data port open: init\r\n");
				break;

			}

    		TcpOpen(&p->TCPopen_1);					/*open a listening socket*/

			/*server connection accepted*/
			if(p->TCPopen_1.status == 0){
				/*NOTE: data port is opened; next: listen for remote connection*/
				DBG("datasocket - open ok\r\n");
 				bgSMSetNextState(psm, bgSMGetState(psm) + 1);
				break;
			}

			/*waiting for connection || pNA is busy*/
			if( (p->TCPopen_1.status == 0xFFFF) ){
				DBG("datasocket - waiting to open socket\r\n");
				break;
			}

			DBG("datasocket - error=%d\r\n", p->TCPopen_1.status);

			bgSMRaiseError(psm, "TCPopen() error", 0, p->TCPopen_1.status);
		break;
		case 2:
			bgSMSetStateName(psm, "DataPort-Init");
			if(bgSMIsStateInit(psm)){
				p->sockData_Timer = 0;

				p->TCPserv_1.enable = 1;            		/* enables the FUB */
				p->TCPserv_1.ident = p->TCPopen_1.ident;    /* ident from open */

	    		p->TCPrecv_1.enable = 1;           	/* enables the FUB */
				p->rxDataBuff = 0;
				p->recvLenData = 0;
				p->TCPrecv_1.datamax = 10000;		/* size of the buffer should be > 8192*/
    			TMP_alloc (p->TCPrecv_1.datamax, (void**)&p->rxDataBuff);   /*allocate memory for data rx*/
	    		p->TCPrecv_1.pData = (UDINT)p->rxDataBuff; /* address of the buffer */
	    		p->TCPclose_1.enable = 1;                  /* enables the FUB */

				DBG("data port open\r\n");
				break;

			}

    		TcpServer(&p->TCPserv_1);					/*listen for a server connection request*/

			/*server connection accepted*/
			if(p->TCPserv_1.status == 0){
				/*NOTE: data port is ready if either connection is accepted or if waiting for connection*/
				DBG("datasocket - connected\r\n");
				p->TCPrecv_1.ident = p->TCPserv_1.identclnt;
				p->TCPclose_1.ident = p->TCPserv_1.identclnt;
				p->isDataPortReady = 1;
 				bgSMSetNextState(psm, bgSMGetState(psm) + 1);
				break;
			}

			/*waiting for connection || pNA is busy*/
			if( (p->TCPserv_1.status == 0xFFFF) ){
				DBG("datasocket - waiting connection\r\n");
				p->isDataPortReady = 1;
				break;
			}

			DBG("datasocket - error=%d\r\n", p->TCPserv_1.status);

			bgSMRaiseError(psm, "TCPserv() error", 0, p->TCPserv_1.status);
		break;
		case 3:
			bgSMSetStateName(psm, "DataPort-Recv");
			/* recv in progress*/
           	TcpRecv(&p->TCPrecv_1);

			/*recv timer*/
            if(p->sockData_Timer && (p->TCPrecv_1.status == 0xFFFF)){
    			p->sockData_TimerCounter++;
				DBG("data port recv() busy; counter=%d\r\n", p->sockData_TimerCounter);
            }

            if(p->TCPrecv_1.status == 0){
				/*test only; inc receive counter*/
				p->counter++;

				/*in case data arrives->copy data to user buffer*/
				if(p->TCPrecv_1.recvlen != 0){

					if(p->user.dataBufferLength < (p->recvLenData + p->TCPrecv_1.recvlen) ){
						DBG("!!!! rxBufferOverflow rxLen=%d > rxBufferSize=%d!!!!\r\n", (int)(p->recvLenData + p->TCPrecv_1.recvlen), (int)p->user.dataBufferLength);
						DBG("!!!! INCREASE USER RX BUFFER SIZE !!!!\r\n");
						/*user supplied buffer is too small!!!*/
						bgSMRaiseError(psm, "Data Buffer Overflow!", 0, bgSMGetState(psm));
						break;
					}

					memcpy( (char*)(p->user.dataBuffer + p->recvLenData), p->rxDataBuff, p->TCPrecv_1.recvlen);
					p->recvLenData += p->TCPrecv_1.recvlen;

					p->sockData_TimerCounter = 0;
				}
				else{
					/*Status == 0 && rxLengt == 0 -> remote peer has closed the connection!!!*/
					bgSMSetNextState(psm, bgSMGetState(psm) + 1);
				}
            }
			else
			if(p->sockData_TimerCounter >= p->sockData_TimerTime){
				/*if receive timer expires, close data socket*/
				bgSMSetNextState(psm, bgSMGetState(psm) + 1);
			}

			DBG("data recv(); rxLen=%d, rxStatus=%d, timer=%d \r\n",
				(int)p->TCPrecv_1.recvlen, (int)p->TCPrecv_1.status, (int)p->sockData_TimerCounter);
		break;
		case 4:
			bgSMSetStateName(psm, "DataPort-Close");
            TcpClose(&p->TCPclose_1);          /* set the socket free */

			if(p->TCPclose_1.status == 0){
				p->isDataPortReady = 0;
				p->sockData_Timer = 0;

				/*terminate rx buffer with 0 -> for strings*/
				p->user.dataBuffer[p->recvLenData] = 0;

				bgSMRaiseDone(psm, 0);
			}

			if( p->rxDataBuff ){
				p->rxDataBuff = 0;
				TMP_free (p->TCPrecv_1.datamax, (void**)p->rxDataBuff);
			}
		break;
		default:
			/*unhandled state*/
			bgSMRaiseError(psm, "unknown state", 0, bgSMGetState(psm));
		break;
	}

	if(bgSMOnError(psm)){
		p->TCPclose_1.ident = p->TCPserv_1.identclnt;    /* copy the  Ident number */
	    TcpClose(&p->TCPclose_1);          				/* set the socket free */
		p->isDataPortReady = 0;

		if( p->rxDataBuff ){
			p->rxDataBuff = 0;
			TMP_free (p->TCPrecv_1.datamax, (void**)p->rxDataBuff);
		}
		/*raise error again for cmd level state machine*/
		bgSMRaiseError(psm, "Data Server Error", 0, 0);
 	}

	if(bgSMOnDone(psm)){

	}
}
/*
========================================================================================
*/
void swapBytesInShort(unsigned short *value)
{

union{
	unsigned short 	shortValue;
	unsigned char	bytes[2];
}swapValue;

unsigned char tempByte;

	swapValue.shortValue = *value;
	tempByte = swapValue.bytes[0];
	swapValue.bytes[0] = swapValue.bytes[1];
	swapValue.bytes[1] = tempByte;
	*value = swapValue.shortValue;
}
/*
========================================================================================
*/
void setSocketAddressData(ETH_sockaddr_typ *adrData, char *hostIpAddressString, unsigned short hostPort)
{

	unsigned short sin_family;
	unsigned short family;
	unsigned short length;
	unsigned short port;

	family = ETH_AF_INET;
	length = sizeof(ETH_sockaddr_typ);
	sin_family = (family << 8) + length;

	adrData->sin_family = sin_family;
	port = hostPort;
	swapBytesInShort(&port);
	adrData->sin_port = port;
	if( strlen(hostIpAddressString) < 8)
		adrData->sin_addr = ETH_INADDR_ANY;
	else
		adrData->sin_addr = inet_addr( (unsigned long) hostIpAddressString);
	adrData->sin_zero[0]=0;
	adrData->sin_zero[1]=0;
	adrData->sin_zero[2]=0;
	adrData->sin_zero[3]=0;
	adrData->sin_zero[4]=0;
	adrData->sin_zero[5]=0;
	adrData->sin_zero[6]=0;
	adrData->sin_zero[7]=0;
}
/*
========================================================================================
========================================================================================
========================================================================================
========================================================================================
*/
/*EOF*/
```

#### bgPVLogger3.c
```c
/********************************************************************
 * COPYRIGHT -- belgor
 ********************************************************************
 * Package: bglib
 * File: bgPVLogger.c
 * Author: goran
 * Created: October 13, 2011
 *******************************************************************/

#include <bur/plctypes.h>
#include <AsDefault.h>

/**
 Simple logging.
 Set to 0 when simple log is not needed
 To view this log, open Automation Studio  watch window and insert below defined
 logxx variable.
 Most recent log entry is always on the top (index 0)
 */
#if 1
//#include "bgsprintf.h"
#include "bgstring.h"

typedef struct bgPVLogger_typ
{
	int initOk;
	char* logbuf;
	int entryCount;
	int entryLen;
}bgPVLogger_typ;

static bgPVLogger_typ lgrObj;	//PV logger object
static bgPVLogger_typ* lgr;	//PV logger object

static void bgPVLoggerInit(bgPVLogger_typ* p, char* logbuf, int logEntryCount, int logEntryLen)
{
	if(!p || !logbuf || !logEntryCount || !logEntryLen)
		return;

	p->logbuf = logbuf;
	p->entryCount = logEntryCount;
	p->entryLen = logEntryLen;
	p->initOk = 1;
}

static void shiftlog(bgPVLogger_typ* p)
{
int ii;
	if(!p || !p->initOk)
		return;

	for(ii=(p->entryCount-2); ii>=0; ii--){
		bgStrCpyN(&p->logbuf[(ii+1) * p->entryLen], &p->logbuf[ii * p->entryLen], p->entryLen);
	}
}

#define DBG(pLoggerInstance, format, args...)	{shiftlog(pLoggerInstance); snprintf2(&pLoggerInstance->logbuf[0], pLoggerInstance->entryLen, format, ## args);}
#define DBGINIT(pLoggerInstance,  logbuf, logEntryCount, logEntryLen) {lgr = &lgrObj; bgPVLoggerInit(pLoggerInstance, &logbuf[0][0], logEntryCount, logEntryLen);}

#else

#define DBG(format, args...)   ;

#endif

//#endif
```
